(* PLC project Untitled3, Machine Expert Logic Builder V20.2.8.0, author Dylan *)
(* stored: creationDateTime 2023-03-14T07:56:13.4423497, version 0.0.0.0, modificationDateTime 2023-03-14T07:50:20.7728171 *)

{attribute 'qualified_only'}
{attribute 'strict'}
TYPE ET_9STATE_MONITORING : (STOPPED := 0, RUNNING := 1, STARTING := 2, STOPPING := 3, START_FAIL := 4, STOP_FAIL := 5, UNEXPECTED_START := 6, UNEXPECTED_STOP := 7, FIRE_STOP := 8, UNKNOWN := 9);
END_TYPE

{attribute 'qualified_only'}
{attribute 'strict'}
TYPE ET_ROOM_STATE : (DEPROX := 0, STANDBY := 1, ALARM := 2, ISOLATE := 3, POSITVE := 4);
END_TYPE

{attribute 'qualified_only'}
{attribute 'strict'}
TYPE ET_ROOM_MODE : (ISOLATION := 0, STANDBY := 1);
END_TYPE

PROGRAM RM59_STATUS
  VAR
    RM_MODE : ET_ROOM_MODE;
    ALARM_DELAY : TON;
    IS_ALARM : BOOL;
    TOF_BUZZER : TOF;
    RM_BUZZER_LOCAL : BOOL;
    IS_LOCAL_ALARM : BOOL;
    FB_ROOM_STATE_0 : FB_ROOM_STATE;
  END_VAR

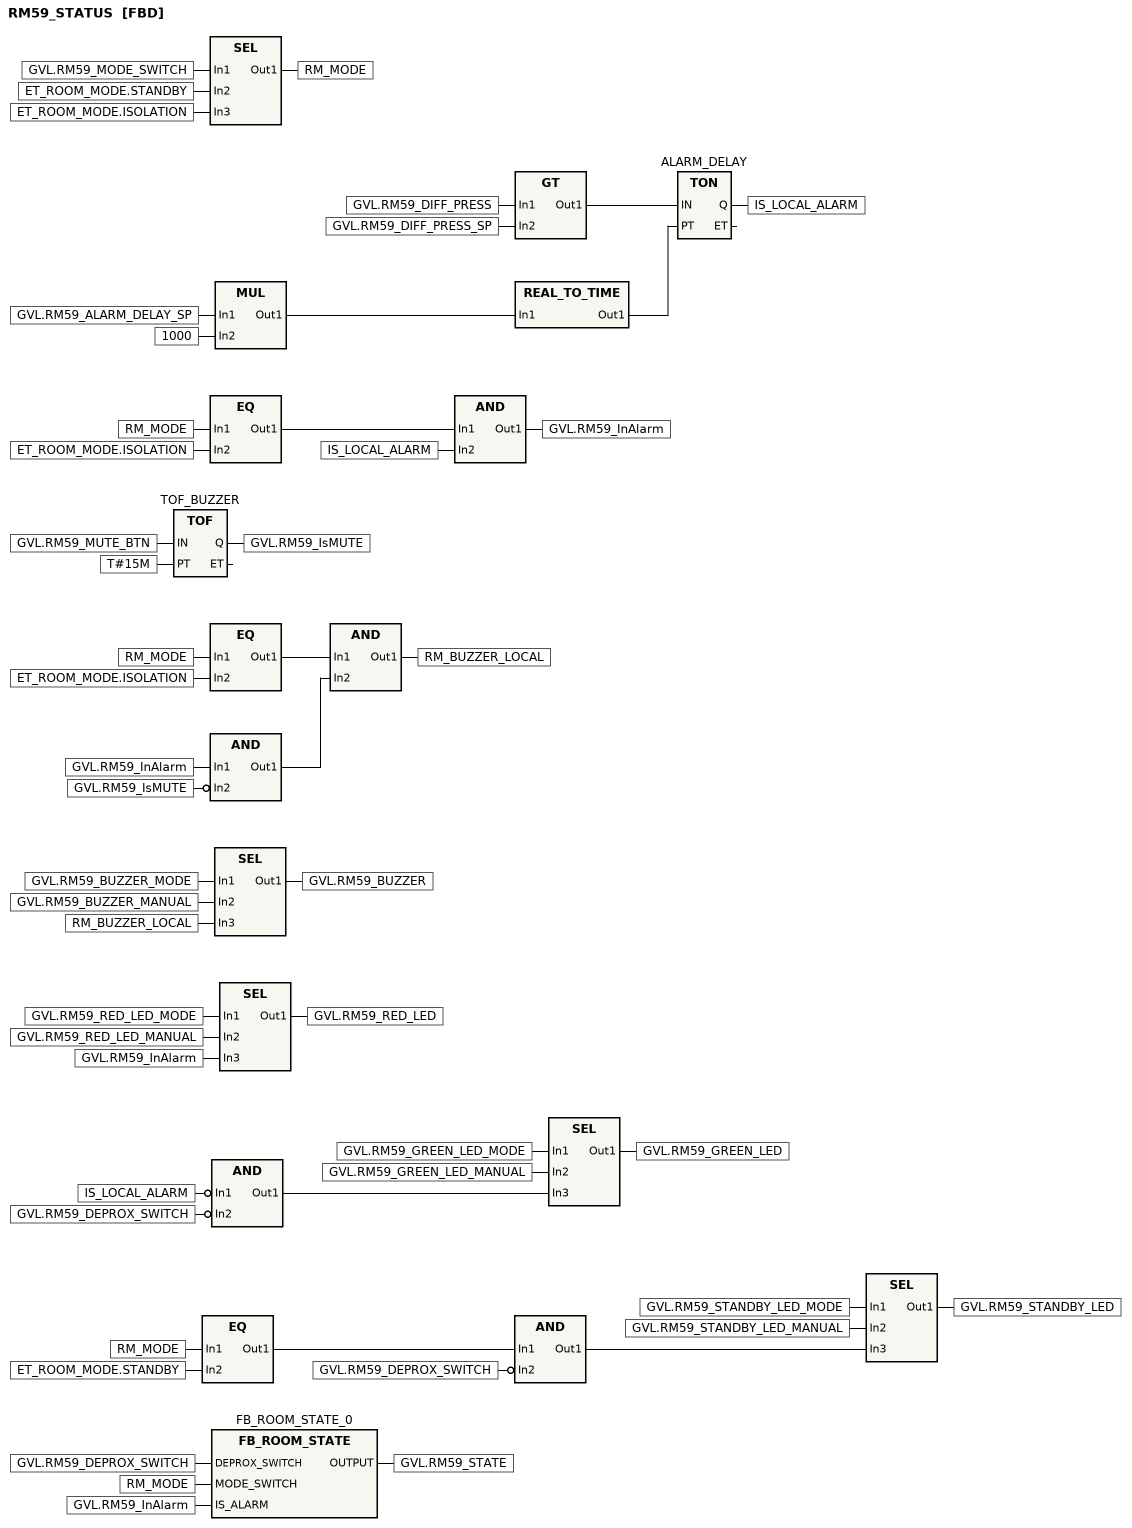
(* FBD diagram, written out as Structured Text *)
(* The mode switch located on the room alarm panel is to switch the room status between isolation mode and standby mode. *)
RM_MODE := SEL(GVL.RM59_MODE_SWITCH, ET_ROOM_MODE.STANDBY, ET_ROOM_MODE.ISOLATION);
(* generate alarms when RM DIFF PRESS >  RM DIFF PRESS SP.
the alarm will show on LED *)
ALARM_DELAY(IN := GVL.RM59_DIFF_PRESS > GVL.RM59_DIFF_PRESS_SP, PT := REAL_TO_TIME(GVL.RM59_ALARM_DELAY_SP * 1000));
IS_LOCAL_ALARM := ALARM_DELAY.Q;
(* ROOM IN ALARM *)
GVL.RM59_InAlarm := RM_MODE = ET_ROOM_MODE.ISOLATION AND IS_LOCAL_ALARM;
(* BUZZER
If the room is operating in isolation mode, the buzzer will activate until the panel RED button is pressed by an operator. If the room pressure remains outside of the acceptable range for a further 15 minutes, then the room buzzer will re-enable.

DISABLE BUZZER *)
TOF_BUZZER(IN := GVL.RM59_MUTE_BTN, PT := T#15M);
GVL.RM59_IsMUTE := TOF_BUZZER.Q;
(* BUZZER
If the room is operating in isolation mode, the buzzer will activate until the panel RED button is pressed by an operator. If the room pressure remains outside of the acceptable range for a further 15 minutes, then the room buzzer will re-enable. *)
RM_BUZZER_LOCAL := RM_MODE = ET_ROOM_MODE.ISOLATION AND GVL.RM59_InAlarm AND NOT GVL.RM59_IsMUTE;
(* AUTO/ MANUAL  MODE FROM BMS / BUZZER *)
GVL.RM59_BUZZER := SEL(GVL.RM59_BUZZER_MODE, GVL.RM59_BUZZER_MANUAL, RM_BUZZER_LOCAL);
(* AUTO/ MANUAL  MODE FROM BMS / RED LED *)
GVL.RM59_RED_LED := SEL(GVL.RM59_RED_LED_MODE, GVL.RM59_RED_LED_MANUAL, GVL.RM59_InAlarm);
(* AUTO/ MANUAL  MODE FROM BMS / GREEN LED *)
GVL.RM59_GREEN_LED := SEL(GVL.RM59_GREEN_LED_MODE, GVL.RM59_GREEN_LED_MANUAL, NOT IS_LOCAL_ALARM AND NOT GVL.RM59_DEPROX_SWITCH);
GVL.RM59_STANDBY_LED := SEL(GVL.RM59_STANDBY_LED_MODE, GVL.RM59_STANDBY_LED_MANUAL, RM_MODE = ET_ROOM_MODE.STANDBY AND NOT GVL.RM59_DEPROX_SWITCH);
(* ROOMT STATUS *)
FB_ROOM_STATE_0(DEPROX_SWITCH := GVL.RM59_DEPROX_SWITCH, MODE_SWITCH := RM_MODE, IS_ALARM := GVL.RM59_InAlarm);
GVL.RM59_STATE := FB_ROOM_STATE_0.OUTPUT;
END_PROGRAM

PROGRAM RM51_DEPROX
  VAR
    ENABLE_BLINKING : BOOL;
    FB_PULSE_GENERATOR_0 : FB_PULSE_GENERATOR;
  END_VAR

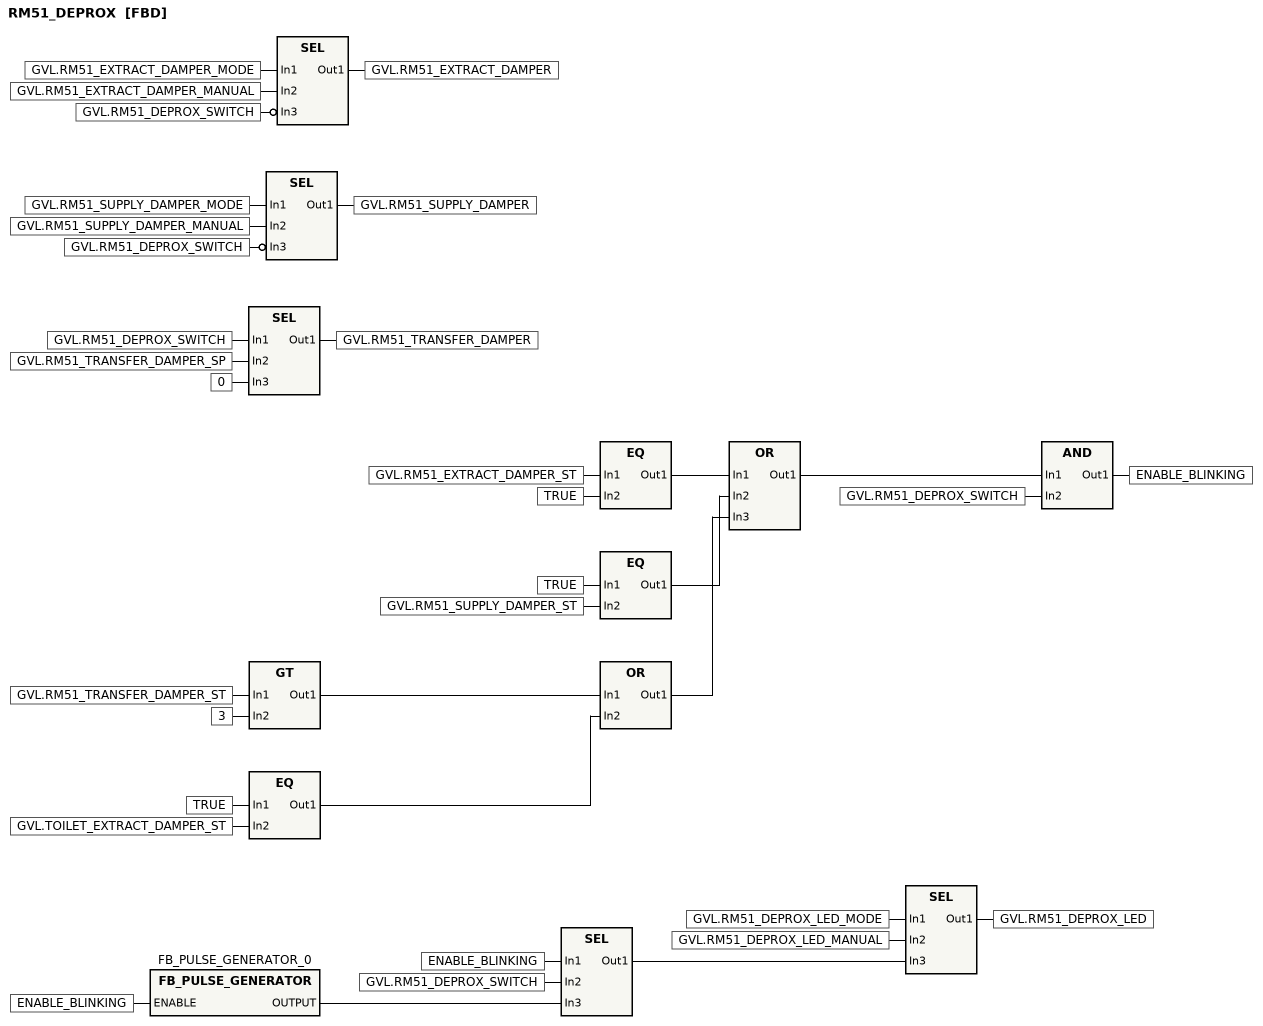
(* FBD diagram, written out as Structured Text *)
(* Return Air Damper - close damper in deprox mode

Deprox Switch. 0=normal 1=deprox *)
GVL.RM51_EXTRACT_DAMPER := SEL(GVL.RM51_EXTRACT_DAMPER_MODE, GVL.RM51_EXTRACT_DAMPER_MANUAL, NOT GVL.RM51_DEPROX_SWITCH);
(* Supply Air Damper - close damper in deprox mode

Deprox Switch. 0=normal 1=deprox *)
GVL.RM51_SUPPLY_DAMPER := SEL(GVL.RM51_SUPPLY_DAMPER_MODE, GVL.RM51_SUPPLY_DAMPER_MANUAL, NOT GVL.RM51_DEPROX_SWITCH);
(* Transfer Damper - close damper in deprox mode

Deprox Switch. 0=normal 1=deprox *)
GVL.RM51_TRANSFER_DAMPER := SEL(GVL.RM51_DEPROX_SWITCH, GVL.RM51_TRANSFER_DAMPER_SP, 0);
(* enable blinking when the room dampers are driving closed *)
ENABLE_BLINKING := (GVL.RM51_EXTRACT_DAMPER_ST = TRUE OR TRUE = GVL.RM51_SUPPLY_DAMPER_ST OR GVL.RM51_TRANSFER_DAMPER_ST > 3 OR TRUE = GVL.TOILET_EXTRACT_DAMPER_ST) AND GVL.RM51_DEPROX_SWITCH;
(* DEPROX LED *)
FB_PULSE_GENERATOR_0(ENABLE := ENABLE_BLINKING);
GVL.RM51_DEPROX_LED := SEL(GVL.RM51_DEPROX_LED_MODE, GVL.RM51_DEPROX_LED_MANUAL, SEL(ENABLE_BLINKING, GVL.RM51_DEPROX_SWITCH, FB_PULSE_GENERATOR_0.OUTPUT));
END_PROGRAM

FUNCTION_BLOCK FB_2STAGES_DUTY
  VAR_INPUT
    isFAN1_FAULT : BOOL;
    isFAN2_FAULT : BOOL;
    STANDBY_FAN : INT := 1;
    FAN_SPD : REAL;
  END_VAR
  VAR_OUTPUT
    FAN1_ENABLE : BOOL;
    FAN2_ENABLE : BOOL;
    FAN1_SPD : REAL;
    FAN2_SPD : REAL;
  END_VAR

                    IF (STANDBY_FAN = 1) THEN
	IF(isFAN2_FAULT) THEN
		FAN1_ENABLE := TRUE;
		FAN1_SPD := FAN_SPD;
	ELSE
		FAN1_ENABLE := FALSE;
		FAN1_SPD := 0.0;
	END_IF;
	FAN2_ENABLE := TRUE;
	FAN2_SPD := FAN_SPD;
ELSIF (STANDBY_FAN = 2) THEN
	IF(isFAN1_FAULT) THEN
		FAN2_ENABLE := TRUE;
		FAN2_SPD := FAN_SPD;
	ELSE
		FAN2_ENABLE := FALSE;
		FAN2_SPD := 0.0;
	END_IF;
	FAN1_ENABLE := TRUE;
	FAN1_SPD := FAN_SPD;
END_IF;

                  
END_FUNCTION_BLOCK

PROGRAM RM119_DEPROX
  VAR
    ENABLE_BLINKING : BOOL;
    FB_PULSE_GENERATOR_0 : FB_PULSE_GENERATOR;
  END_VAR

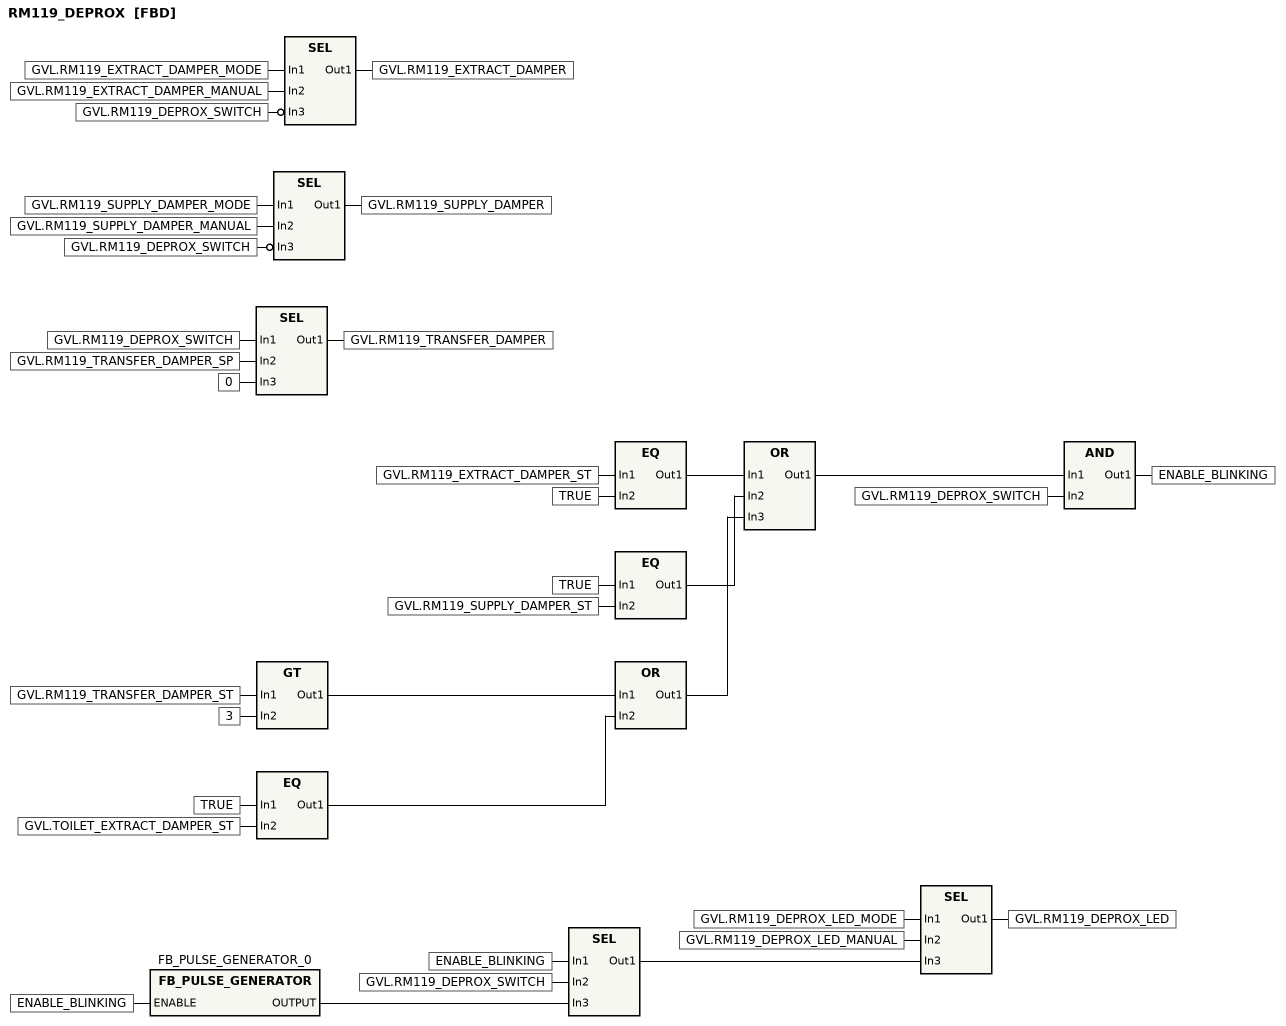
(* FBD diagram, written out as Structured Text *)
(* Return Air Damper - close damper in deprox mode

Deprox Switch. 0=normal 1=deprox *)
GVL.RM119_EXTRACT_DAMPER := SEL(GVL.RM119_EXTRACT_DAMPER_MODE, GVL.RM119_EXTRACT_DAMPER_MANUAL, NOT GVL.RM119_DEPROX_SWITCH);
(* Supply Air Damper - close damper in deprox mode

Deprox Switch. 0=normal 1=deprox *)
GVL.RM119_SUPPLY_DAMPER := SEL(GVL.RM119_SUPPLY_DAMPER_MODE, GVL.RM119_SUPPLY_DAMPER_MANUAL, NOT GVL.RM119_DEPROX_SWITCH);
(* Transfer Damper - close damper in deprox mode

Deprox Switch. 0=normal 1=deprox *)
GVL.RM119_TRANSFER_DAMPER := SEL(GVL.RM119_DEPROX_SWITCH, GVL.RM119_TRANSFER_DAMPER_SP, 0);
(* enable blinking when the room dampers are driving closed *)
ENABLE_BLINKING := (GVL.RM119_EXTRACT_DAMPER_ST = TRUE OR TRUE = GVL.RM119_SUPPLY_DAMPER_ST OR GVL.RM119_TRANSFER_DAMPER_ST > 3 OR TRUE = GVL.TOILET_EXTRACT_DAMPER_ST) AND GVL.RM119_DEPROX_SWITCH;
(* DEPROX LED *)
FB_PULSE_GENERATOR_0(ENABLE := ENABLE_BLINKING);
GVL.RM119_DEPROX_LED := SEL(GVL.RM119_DEPROX_LED_MODE, GVL.RM119_DEPROX_LED_MANUAL, SEL(ENABLE_BLINKING, GVL.RM119_DEPROX_SWITCH, FB_PULSE_GENERATOR_0.OUTPUT));
END_PROGRAM

FUNCTION_BLOCK FB_DUTYTRIGGER
  VAR_INPUT
    INPUT : BOOL;
    MAX_STAGE : INT := 2;
    CURRENT_STAGE : INT;
  END_VAR
  VAR_OUTPUT
    RESULT : INT;
  END_VAR

                    IF(INPUT) THEN
	RESULT := CURRENT_STAGE + 1;
END_IF;

IF(RESULT > MAX_STAGE) OR (RESULT <= 0) THEN
	RESULT:= 1;
END_IF;


                  
END_FUNCTION_BLOCK

PROGRAM RM52_DEPROX
  VAR
    ENABLE_BLINKING : BOOL;
    FB_PULSE_GENERATOR_0 : FB_PULSE_GENERATOR;
  END_VAR

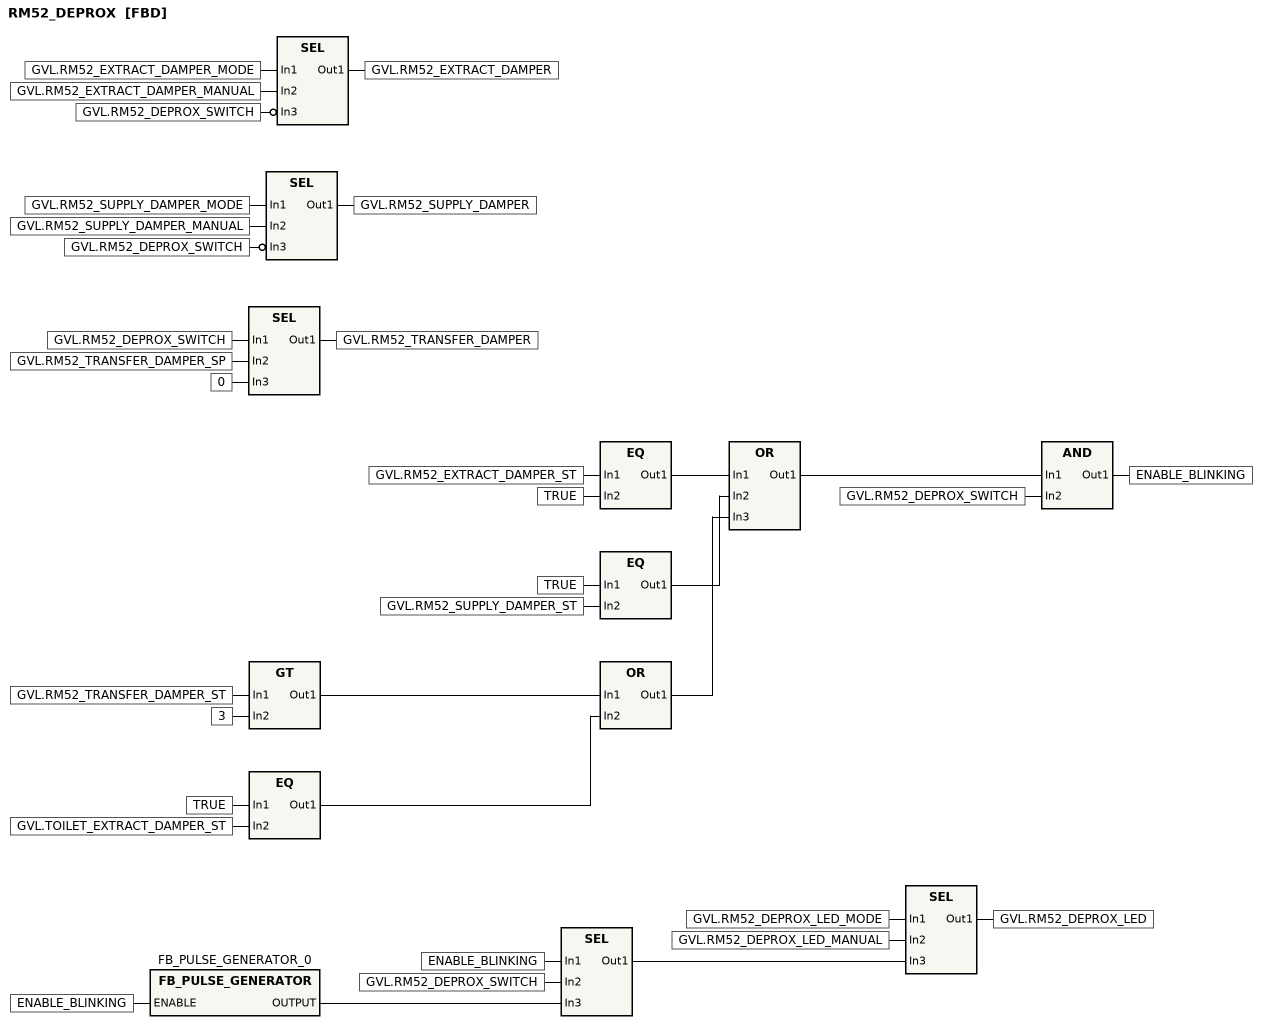
(* FBD diagram, written out as Structured Text *)
(* Return Air Damper - close damper in deprox mode

Deprox Switch. 0=normal 1=deprox *)
GVL.RM52_EXTRACT_DAMPER := SEL(GVL.RM52_EXTRACT_DAMPER_MODE, GVL.RM52_EXTRACT_DAMPER_MANUAL, NOT GVL.RM52_DEPROX_SWITCH);
(* Supply Air Damper - close damper in deprox mode

Deprox Switch. 0=normal 1=deprox *)
GVL.RM52_SUPPLY_DAMPER := SEL(GVL.RM52_SUPPLY_DAMPER_MODE, GVL.RM52_SUPPLY_DAMPER_MANUAL, NOT GVL.RM52_DEPROX_SWITCH);
(* Transfer Damper - close damper in deprox mode

Deprox Switch. 0=normal 1=deprox *)
GVL.RM52_TRANSFER_DAMPER := SEL(GVL.RM52_DEPROX_SWITCH, GVL.RM52_TRANSFER_DAMPER_SP, 0);
(* enable blinking when the room dampers are driving closed *)
ENABLE_BLINKING := (GVL.RM52_EXTRACT_DAMPER_ST = TRUE OR TRUE = GVL.RM52_SUPPLY_DAMPER_ST OR GVL.RM52_TRANSFER_DAMPER_ST > 3 OR TRUE = GVL.TOILET_EXTRACT_DAMPER_ST) AND GVL.RM52_DEPROX_SWITCH;
(* DEPROX LED *)
FB_PULSE_GENERATOR_0(ENABLE := ENABLE_BLINKING);
GVL.RM52_DEPROX_LED := SEL(GVL.RM52_DEPROX_LED_MODE, GVL.RM52_DEPROX_LED_MANUAL, SEL(ENABLE_BLINKING, GVL.RM52_DEPROX_SWITCH, FB_PULSE_GENERATOR_0.OUTPUT));
END_PROGRAM

PROGRAM RM53_DEPROX
  VAR
    ENABLE_BLINKING : BOOL;
    FB_PULSE_GENERATOR_0 : FB_PULSE_GENERATOR;
  END_VAR

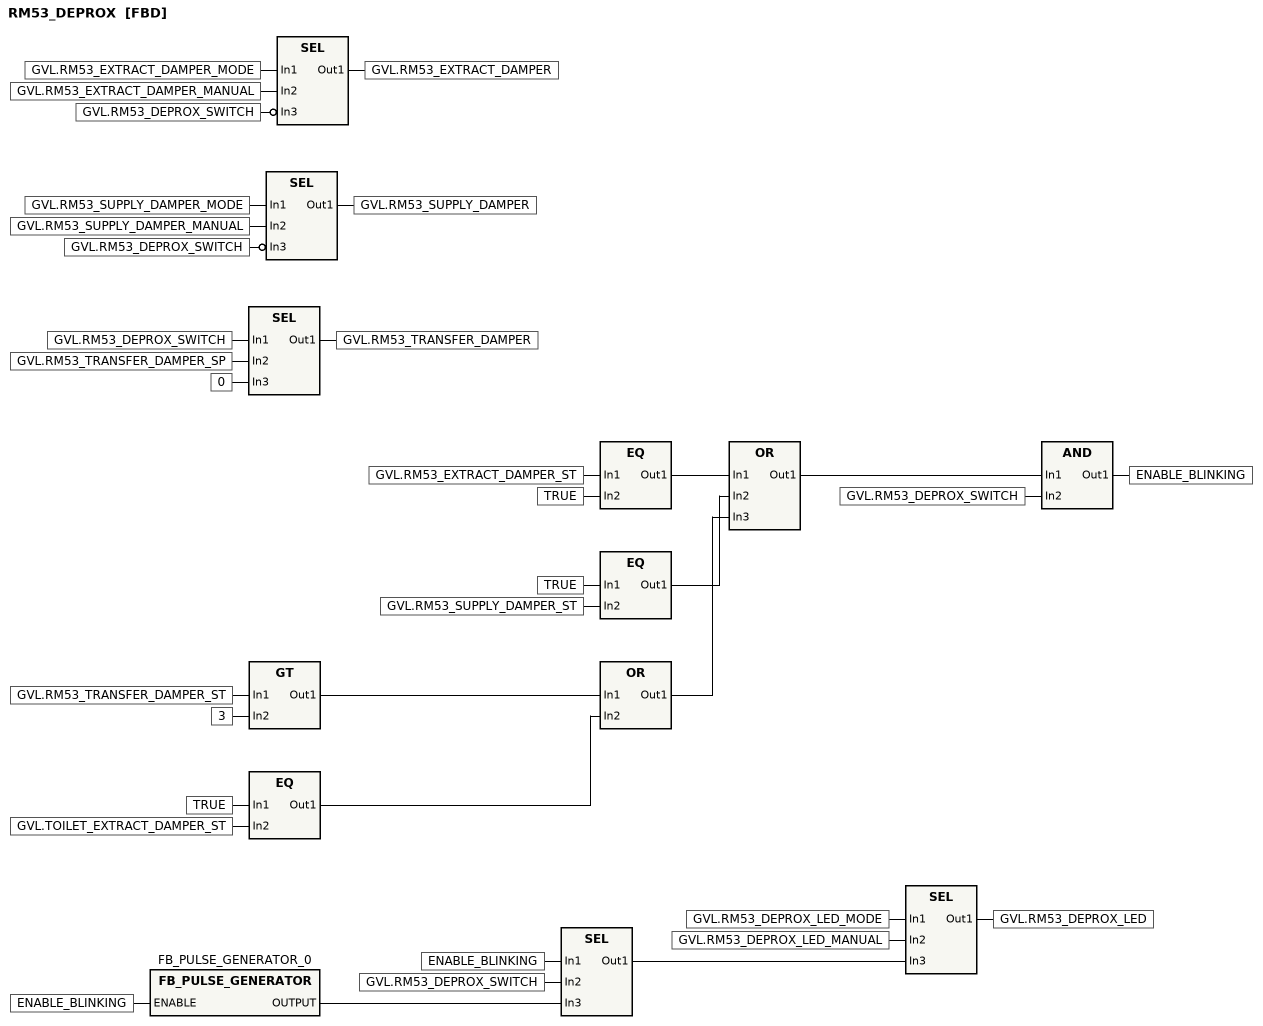
(* FBD diagram, written out as Structured Text *)
(* Return Air Damper - close damper in deprox mode

Deprox Switch. 0=normal 1=deprox *)
GVL.RM53_EXTRACT_DAMPER := SEL(GVL.RM53_EXTRACT_DAMPER_MODE, GVL.RM53_EXTRACT_DAMPER_MANUAL, NOT GVL.RM53_DEPROX_SWITCH);
(* Supply Air Damper - close damper in deprox mode

Deprox Switch. 0=normal 1=deprox *)
GVL.RM53_SUPPLY_DAMPER := SEL(GVL.RM53_SUPPLY_DAMPER_MODE, GVL.RM53_SUPPLY_DAMPER_MANUAL, NOT GVL.RM53_DEPROX_SWITCH);
(* Transfer Damper - close damper in deprox mode

Deprox Switch. 0=normal 1=deprox *)
GVL.RM53_TRANSFER_DAMPER := SEL(GVL.RM53_DEPROX_SWITCH, GVL.RM53_TRANSFER_DAMPER_SP, 0);
(* enable blinking when the room dampers are driving closed *)
ENABLE_BLINKING := (GVL.RM53_EXTRACT_DAMPER_ST = TRUE OR TRUE = GVL.RM53_SUPPLY_DAMPER_ST OR GVL.RM53_TRANSFER_DAMPER_ST > 3 OR TRUE = GVL.TOILET_EXTRACT_DAMPER_ST) AND GVL.RM53_DEPROX_SWITCH;
(* DEPROX LED *)
FB_PULSE_GENERATOR_0(ENABLE := ENABLE_BLINKING);
GVL.RM53_DEPROX_LED := SEL(GVL.RM53_DEPROX_LED_MODE, GVL.RM53_DEPROX_LED_MANUAL, SEL(ENABLE_BLINKING, GVL.RM53_DEPROX_SWITCH, FB_PULSE_GENERATOR_0.OUTPUT));
END_PROGRAM

FUNCTION_BLOCK FB_3STAGES_DUTY
  VAR_INPUT
    isFAN1_FAULT : BOOL;
    isFAN2_FAULT : BOOL;
    isFAN3_FAULT : BOOL;
    STANDBY_FAN : INT := 1;
    FAN_SPD : REAL;
  END_VAR
  VAR_OUTPUT
    FAN1_ENABLE : BOOL;
    FAN2_ENABLE : BOOL;
    FAN3_ENABLE : BOOL;
    FAN1_SPD : REAL;
    FAN2_SPD : REAL;
    FAN3_SPD : REAL;
  END_VAR

                    IF (STANDBY_FAN = 1) THEN
	IF(isFAN2_FAULT OR isFAN3_FAULT) THEN
		FAN1_ENABLE := TRUE;
		FAN1_SPD := FAN_SPD;
	ELSE
		FAN1_ENABLE := FALSE;
		FAN1_SPD := 0.0;
	END_IF;
	FAN2_ENABLE := TRUE;
	FAN3_ENABLE := TRUE;
	FAN2_SPD := FAN_SPD;
	FAN3_SPD := FAN_SPD;
ELSIF (STANDBY_FAN = 2) THEN
	IF(isFAN1_FAULT OR isFAN3_FAULT) THEN
		FAN2_ENABLE := TRUE;
		FAN2_SPD := FAN_SPD;
	ELSE
		FAN2_ENABLE := FALSE;
		FAN2_SPD := 0.0;
	END_IF;
	FAN1_ENABLE := TRUE;
	FAN3_ENABLE := TRUE;
	FAN1_SPD := FAN_SPD;
	FAN3_SPD := FAN_SPD;
ELSIF (STANDBY_FAN = 3) THEN
	IF(isFAN1_FAULT OR isFAN2_FAULT) THEN
		FAN3_ENABLE := TRUE;
		FAN3_SPD := FAN_SPD;
	ELSE
		FAN3_ENABLE := FALSE;
		FAN3_SPD := 0.0;
	END_IF;
	FAN1_ENABLE := TRUE;
	FAN2_ENABLE := TRUE;
	FAN1_SPD := FAN_SPD;
	FAN2_SPD := FAN_SPD;
END_IF;

                  
END_FUNCTION_BLOCK

PROGRAM RM119_STATUS
  VAR
    RM_MODE : ET_ROOM_MODE;
    ALARM_DELAY : TON;
    IS_ALARM : BOOL;
    TOF_BUZZER : TOF;
    RM_BUZZER_LOCAL : BOOL;
    IS_LOCAL_ALARM : BOOL;
    FB_ROOM_STATE_0 : FB_ROOM_STATE;
  END_VAR

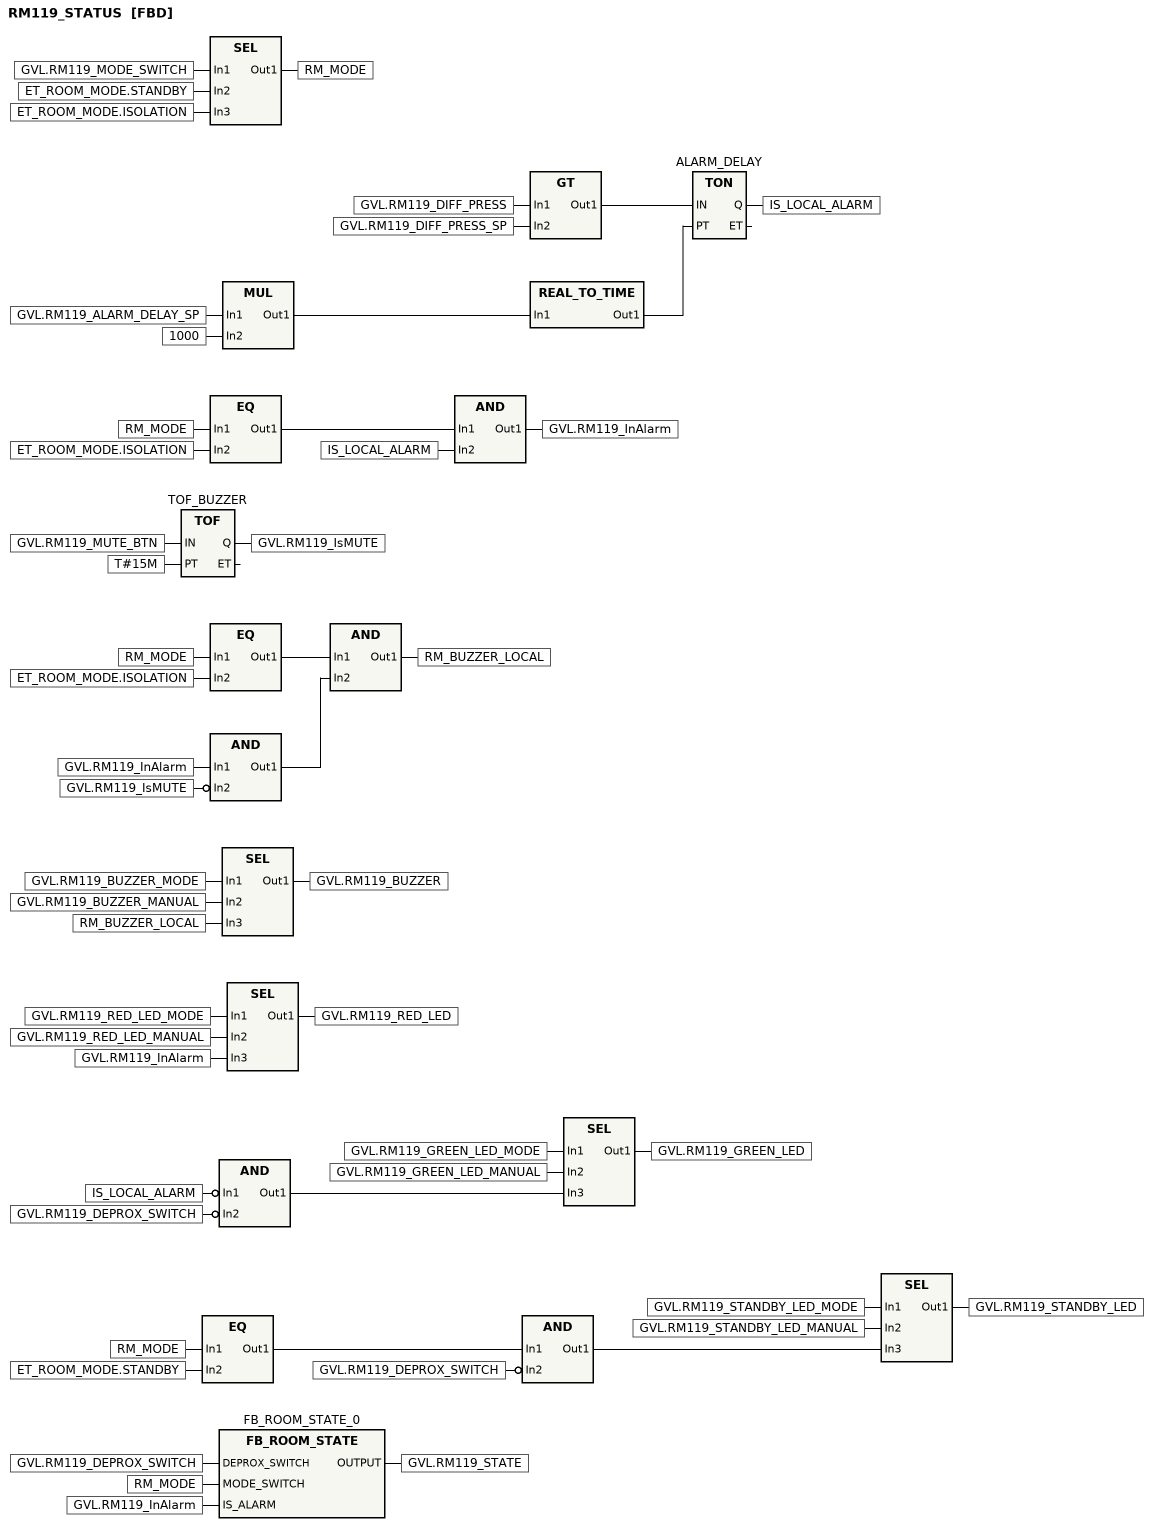
(* FBD diagram, written out as Structured Text *)
(* The mode switch located on the room alarm panel is to switch the room status between isolation mode and standby mode. *)
RM_MODE := SEL(GVL.RM119_MODE_SWITCH, ET_ROOM_MODE.STANDBY, ET_ROOM_MODE.ISOLATION);
(* generate alarms when RM DIFF PRESS >  RM DIFF PRESS SP.
the alarm will show on LED *)
ALARM_DELAY(IN := GVL.RM119_DIFF_PRESS > GVL.RM119_DIFF_PRESS_SP, PT := REAL_TO_TIME(GVL.RM119_ALARM_DELAY_SP * 1000));
IS_LOCAL_ALARM := ALARM_DELAY.Q;
(* ROOM IN ALARM *)
GVL.RM119_InAlarm := RM_MODE = ET_ROOM_MODE.ISOLATION AND IS_LOCAL_ALARM;
(* BUZZER
If the room is operating in isolation mode, the buzzer will activate until the panel RED button is pressed by an operator. If the room pressure remains outside of the acceptable range for a further 15 minutes, then the room buzzer will re-enable.

DISABLE BUZZER *)
TOF_BUZZER(IN := GVL.RM119_MUTE_BTN, PT := T#15M);
GVL.RM119_IsMUTE := TOF_BUZZER.Q;
(* BUZZER
If the room is operating in isolation mode, the buzzer will activate until the panel RED button is pressed by an operator. If the room pressure remains outside of the acceptable range for a further 15 minutes, then the room buzzer will re-enable. *)
RM_BUZZER_LOCAL := RM_MODE = ET_ROOM_MODE.ISOLATION AND GVL.RM119_InAlarm AND NOT GVL.RM119_IsMUTE;
(* AUTO/ MANUAL  MODE FROM BMS / BUZZER *)
GVL.RM119_BUZZER := SEL(GVL.RM119_BUZZER_MODE, GVL.RM119_BUZZER_MANUAL, RM_BUZZER_LOCAL);
(* AUTO/ MANUAL  MODE FROM BMS / RED LED *)
GVL.RM119_RED_LED := SEL(GVL.RM119_RED_LED_MODE, GVL.RM119_RED_LED_MANUAL, GVL.RM119_InAlarm);
(* AUTO/ MANUAL  MODE FROM BMS / GREEN LED *)
GVL.RM119_GREEN_LED := SEL(GVL.RM119_GREEN_LED_MODE, GVL.RM119_GREEN_LED_MANUAL, NOT IS_LOCAL_ALARM AND NOT GVL.RM119_DEPROX_SWITCH);
GVL.RM119_STANDBY_LED := SEL(GVL.RM119_STANDBY_LED_MODE, GVL.RM119_STANDBY_LED_MANUAL, RM_MODE = ET_ROOM_MODE.STANDBY AND NOT GVL.RM119_DEPROX_SWITCH);
(* ROOMT STATUS *)
FB_ROOM_STATE_0(DEPROX_SWITCH := GVL.RM119_DEPROX_SWITCH, MODE_SWITCH := RM_MODE, IS_ALARM := GVL.RM119_InAlarm);
GVL.RM119_STATE := FB_ROOM_STATE_0.OUTPUT;
END_PROGRAM

PROGRAM RM71_DEPROX
  VAR
    ENABLE_BLINKING : BOOL;
    FB_PULSE_GENERATOR_0 : FB_PULSE_GENERATOR;
  END_VAR

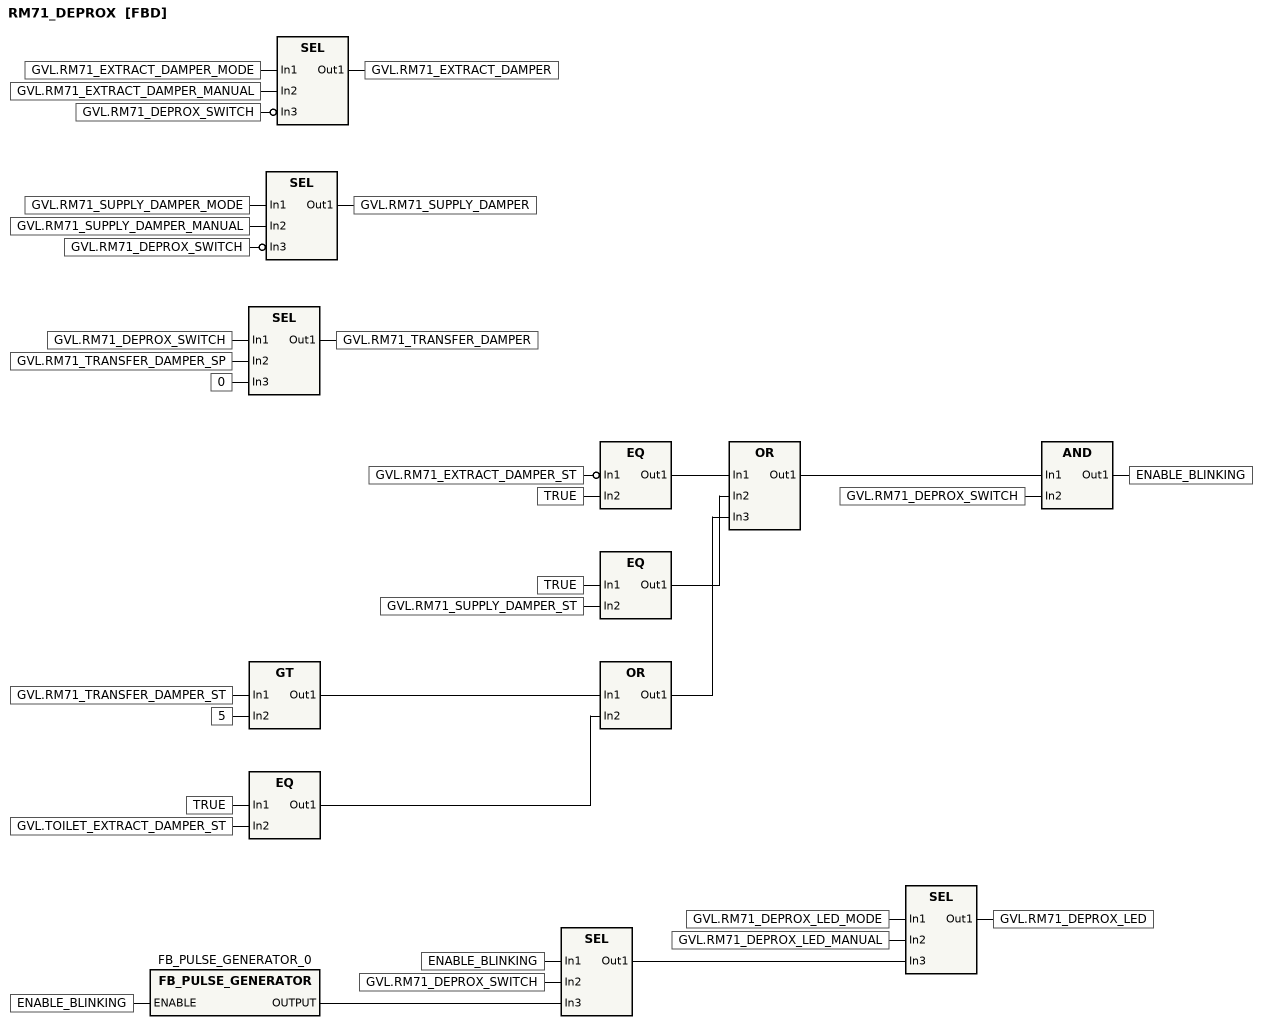
(* FBD diagram, written out as Structured Text *)
(* Return Air Damper - close damper in deprox mode

Deprox Switch. 0=normal 1=deprox *)
GVL.RM71_EXTRACT_DAMPER := SEL(GVL.RM71_EXTRACT_DAMPER_MODE, GVL.RM71_EXTRACT_DAMPER_MANUAL, NOT GVL.RM71_DEPROX_SWITCH);
(* Supply Air Damper - close damper in deprox mode

Deprox Switch. 0=normal 1=deprox *)
GVL.RM71_SUPPLY_DAMPER := SEL(GVL.RM71_SUPPLY_DAMPER_MODE, GVL.RM71_SUPPLY_DAMPER_MANUAL, NOT GVL.RM71_DEPROX_SWITCH);
(* Transfer Damper - close damper in deprox mode

Deprox Switch. 0=normal 1=deprox *)
GVL.RM71_TRANSFER_DAMPER := SEL(GVL.RM71_DEPROX_SWITCH, GVL.RM71_TRANSFER_DAMPER_SP, 0);
(* enable blinking when the room dampers are driving closed *)
ENABLE_BLINKING := (NOT GVL.RM71_EXTRACT_DAMPER_ST = TRUE OR TRUE = GVL.RM71_SUPPLY_DAMPER_ST OR GVL.RM71_TRANSFER_DAMPER_ST > 5 OR TRUE = GVL.TOILET_EXTRACT_DAMPER_ST) AND GVL.RM71_DEPROX_SWITCH;
(* DEPROX LED *)
FB_PULSE_GENERATOR_0(ENABLE := ENABLE_BLINKING);
GVL.RM71_DEPROX_LED := SEL(GVL.RM71_DEPROX_LED_MODE, GVL.RM71_DEPROX_LED_MANUAL, SEL(ENABLE_BLINKING, GVL.RM71_DEPROX_SWITCH, FB_PULSE_GENERATOR_0.OUTPUT));
END_PROGRAM

FUNCTION_BLOCK FB_0_10V_TO_2_10V_OUTPUT
  VAR_OUTPUT
    OUT_PRCT : REAL;  (* 0-10V = 0-100% *)
  END_VAR
  VAR_INPUT
    IN_PRCT : REAL;  (* 2-10V = 0-100% *)
  END_VAR

                    OUT_PRCT := ((IN_PRCT * 0.08) + 2) * 10;
                  
END_FUNCTION_BLOCK

PROGRAM RM52_STATUS
  VAR
    RM_MODE : ET_ROOM_MODE;
    ALARM_DELAY : TON;
    IS_ALARM : BOOL;
    TOF_BUZZER : TOF;
    RM_BUZZER_LOCAL : BOOL;
    IS_LOCAL_ALARM : BOOL;
    FB_ROOM_STATE_0 : FB_ROOM_STATE;
  END_VAR

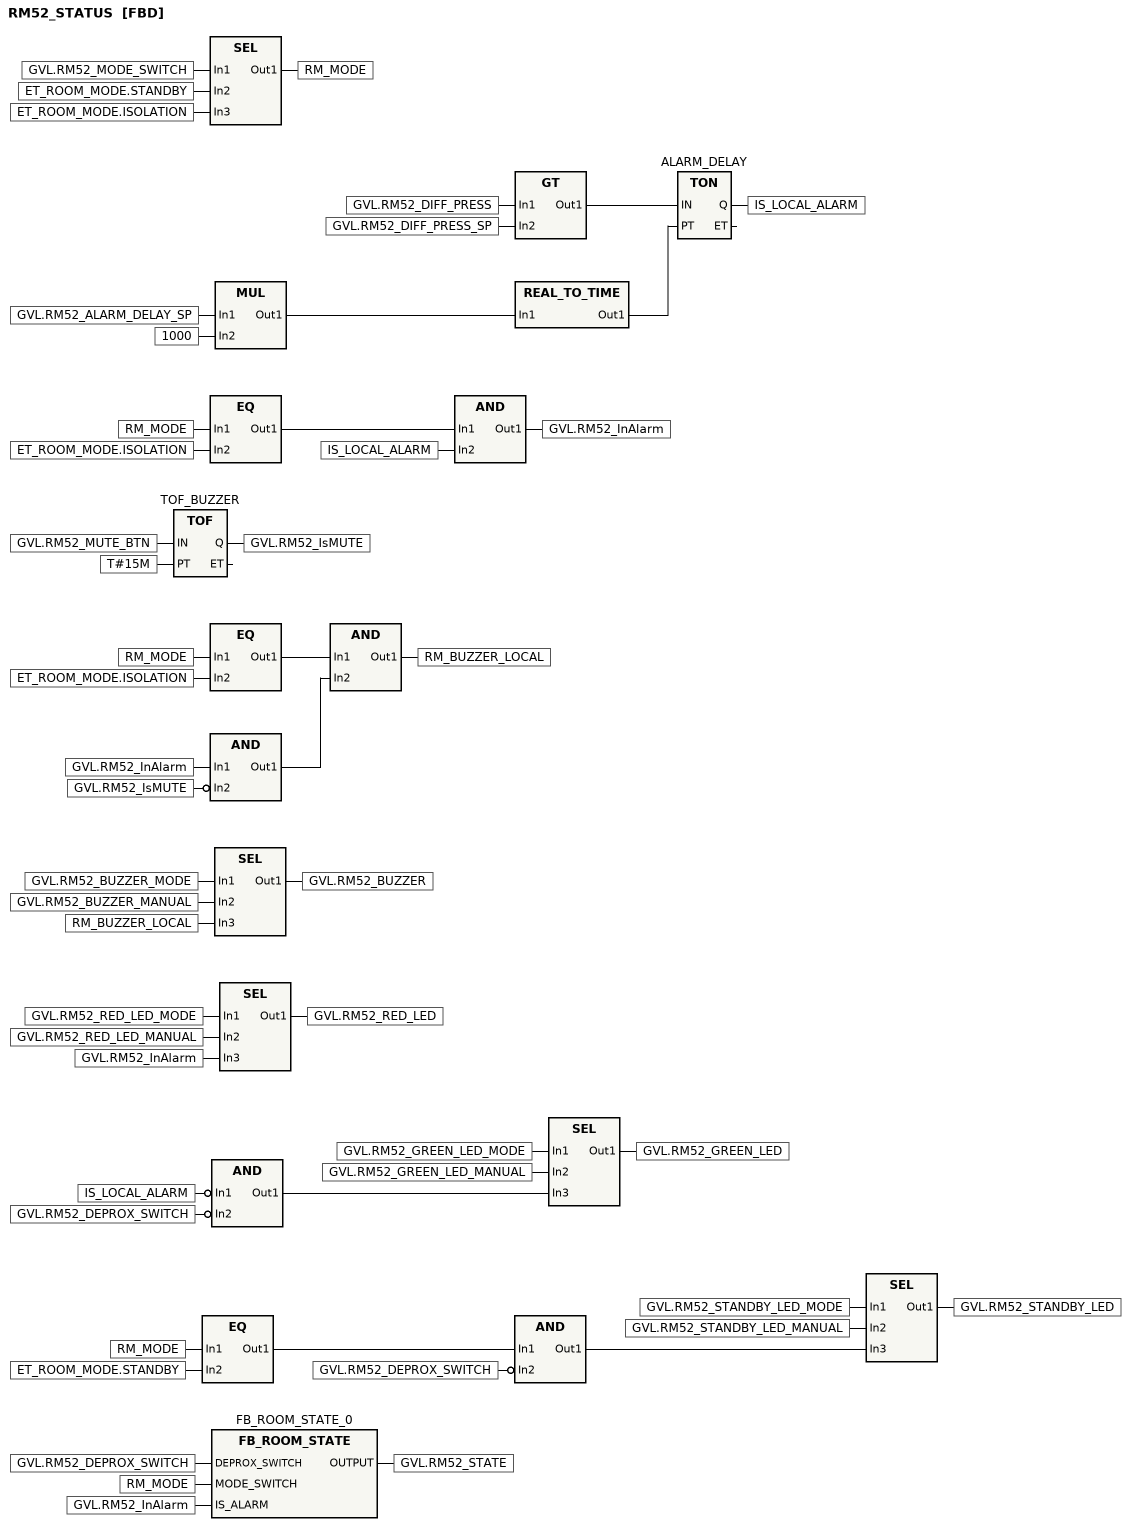
(* FBD diagram, written out as Structured Text *)
(* The mode switch located on the room alarm panel is to switch the room status between isolation mode and standby mode. *)
RM_MODE := SEL(GVL.RM52_MODE_SWITCH, ET_ROOM_MODE.STANDBY, ET_ROOM_MODE.ISOLATION);
(* generate alarms when RM DIFF PRESS >  RM DIFF PRESS SP.
the alarm will show on LED *)
ALARM_DELAY(IN := GVL.RM52_DIFF_PRESS > GVL.RM52_DIFF_PRESS_SP, PT := REAL_TO_TIME(GVL.RM52_ALARM_DELAY_SP * 1000));
IS_LOCAL_ALARM := ALARM_DELAY.Q;
(* ROOM IN ALARM *)
GVL.RM52_InAlarm := RM_MODE = ET_ROOM_MODE.ISOLATION AND IS_LOCAL_ALARM;
(* BUZZER
If the room is operating in isolation mode, the buzzer will activate until the panel RED button is pressed by an operator. If the room pressure remains outside of the acceptable range for a further 15 minutes, then the room buzzer will re-enable.

DISABLE BUZZER *)
TOF_BUZZER(IN := GVL.RM52_MUTE_BTN, PT := T#15M);
GVL.RM52_IsMUTE := TOF_BUZZER.Q;
(* BUZZER
If the room is operating in isolation mode, the buzzer will activate until the panel RED button is pressed by an operator. If the room pressure remains outside of the acceptable range for a further 15 minutes, then the room buzzer will re-enable. *)
RM_BUZZER_LOCAL := RM_MODE = ET_ROOM_MODE.ISOLATION AND GVL.RM52_InAlarm AND NOT GVL.RM52_IsMUTE;
(* AUTO/ MANUAL  MODE FROM BMS / BUZZER *)
GVL.RM52_BUZZER := SEL(GVL.RM52_BUZZER_MODE, GVL.RM52_BUZZER_MANUAL, RM_BUZZER_LOCAL);
(* AUTO/ MANUAL  MODE FROM BMS / RED LED *)
GVL.RM52_RED_LED := SEL(GVL.RM52_RED_LED_MODE, GVL.RM52_RED_LED_MANUAL, GVL.RM52_InAlarm);
(* AUTO/ MANUAL  MODE FROM BMS / GREEN LED *)
GVL.RM52_GREEN_LED := SEL(GVL.RM52_GREEN_LED_MODE, GVL.RM52_GREEN_LED_MANUAL, NOT IS_LOCAL_ALARM AND NOT GVL.RM52_DEPROX_SWITCH);
GVL.RM52_STANDBY_LED := SEL(GVL.RM52_STANDBY_LED_MODE, GVL.RM52_STANDBY_LED_MANUAL, RM_MODE = ET_ROOM_MODE.STANDBY AND NOT GVL.RM52_DEPROX_SWITCH);
(* ROOMT STATUS *)
FB_ROOM_STATE_0(DEPROX_SWITCH := GVL.RM52_DEPROX_SWITCH, MODE_SWITCH := RM_MODE, IS_ALARM := GVL.RM52_InAlarm);
GVL.RM52_STATE := FB_ROOM_STATE_0.OUTPUT;
END_PROGRAM

PROGRAM RM44_3_STATUS
  VAR
    RM_MODE : ET_ROOM_MODE;
    ALARM_DELAY : TON;
    IS_ALARM : BOOL;
    TOF_BUZZER : TOF;
    RM_BUZZER_LOCAL : BOOL;
    IS_LOCAL_ALARM : BOOL;
    FB_ROOM_STATE_0 : FB_ROOM_STATE;
  END_VAR

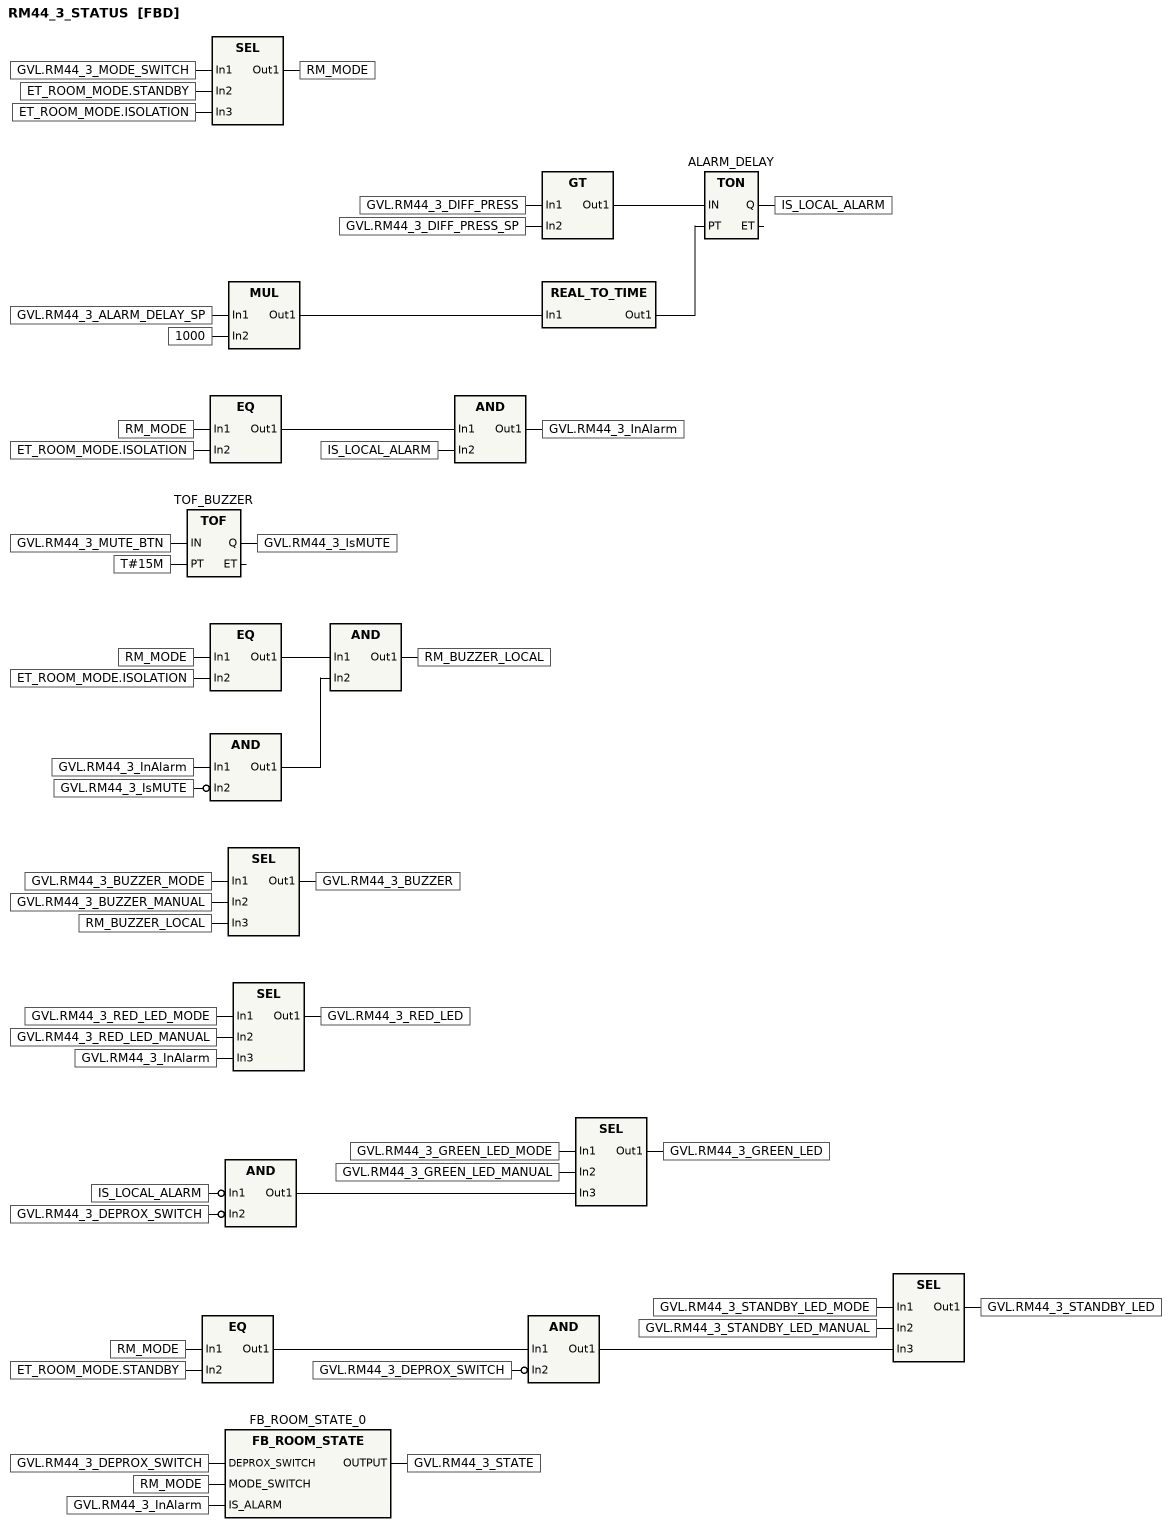
(* FBD diagram, written out as Structured Text *)
(* The mode switch located on the room alarm panel is to switch the room status between isolation mode and standby mode. *)
RM_MODE := SEL(GVL.RM44_3_MODE_SWITCH, ET_ROOM_MODE.STANDBY, ET_ROOM_MODE.ISOLATION);
(* generate alarms when RM DIFF PRESS >  RM DIFF PRESS SP.
the alarm will show on LED *)
ALARM_DELAY(IN := GVL.RM44_3_DIFF_PRESS > GVL.RM44_3_DIFF_PRESS_SP, PT := REAL_TO_TIME(GVL.RM44_3_ALARM_DELAY_SP * 1000));
IS_LOCAL_ALARM := ALARM_DELAY.Q;
(* ROOM IN ALARM *)
GVL.RM44_3_InAlarm := RM_MODE = ET_ROOM_MODE.ISOLATION AND IS_LOCAL_ALARM;
(* BUZZER
If the room is operating in isolation mode, the buzzer will activate until the panel RED button is pressed by an operator. If the room pressure remains outside of the acceptable range for a further 15 minutes, then the room buzzer will re-enable.

DISABLE BUZZER *)
TOF_BUZZER(IN := GVL.RM44_3_MUTE_BTN, PT := T#15M);
GVL.RM44_3_IsMUTE := TOF_BUZZER.Q;
(* BUZZER
If the room is operating in isolation mode, the buzzer will activate until the panel RED button is pressed by an operator. If the room pressure remains outside of the acceptable range for a further 15 minutes, then the room buzzer will re-enable. *)
RM_BUZZER_LOCAL := RM_MODE = ET_ROOM_MODE.ISOLATION AND GVL.RM44_3_InAlarm AND NOT GVL.RM44_3_IsMUTE;
(* AUTO/ MANUAL  MODE FROM BMS / BUZZER *)
GVL.RM44_3_BUZZER := SEL(GVL.RM44_3_BUZZER_MODE, GVL.RM44_3_BUZZER_MANUAL, RM_BUZZER_LOCAL);
(* AUTO/ MANUAL  MODE FROM BMS / RED LED *)
GVL.RM44_3_RED_LED := SEL(GVL.RM44_3_RED_LED_MODE, GVL.RM44_3_RED_LED_MANUAL, GVL.RM44_3_InAlarm);
(* AUTO/ MANUAL  MODE FROM BMS / GREEN LED *)
GVL.RM44_3_GREEN_LED := SEL(GVL.RM44_3_GREEN_LED_MODE, GVL.RM44_3_GREEN_LED_MANUAL, NOT IS_LOCAL_ALARM AND NOT GVL.RM44_3_DEPROX_SWITCH);
GVL.RM44_3_STANDBY_LED := SEL(GVL.RM44_3_STANDBY_LED_MODE, GVL.RM44_3_STANDBY_LED_MANUAL, RM_MODE = ET_ROOM_MODE.STANDBY AND NOT GVL.RM44_3_DEPROX_SWITCH);
(* ROOMT STATUS *)
FB_ROOM_STATE_0(DEPROX_SWITCH := GVL.RM44_3_DEPROX_SWITCH, MODE_SWITCH := RM_MODE, IS_ALARM := GVL.RM44_3_InAlarm);
GVL.RM44_3_STATE := FB_ROOM_STATE_0.OUTPUT;
END_PROGRAM

PROGRAM RM51_STATUS
  VAR
    RM_MODE : ET_ROOM_MODE;
    ALARM_DELAY : TON;
    IS_ALARM : BOOL;
    TOF_BUZZER : TOF;
    RM_BUZZER_LOCAL : BOOL;
    IS_LOCAL_ALARM : BOOL;
    FB_ROOM_STATE_0 : FB_ROOM_STATE;
  END_VAR

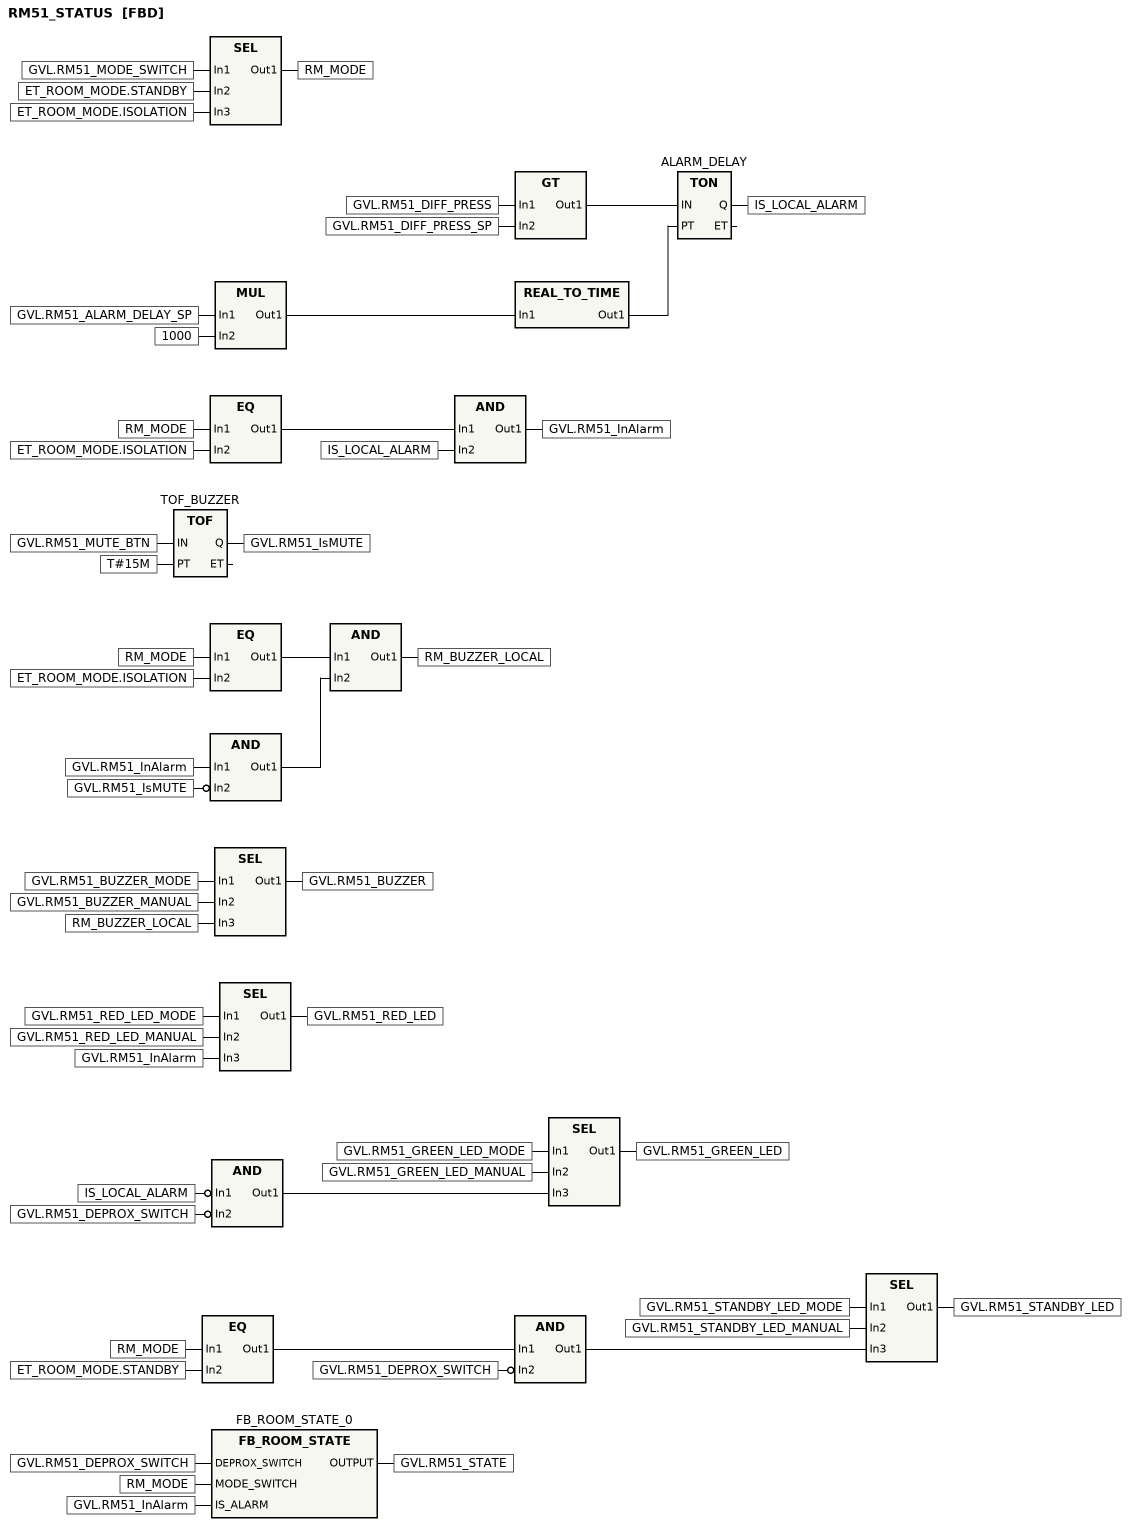
(* FBD diagram, written out as Structured Text *)
(* The mode switch located on the room alarm panel is to switch the room status between isolation mode and standby mode. *)
RM_MODE := SEL(GVL.RM51_MODE_SWITCH, ET_ROOM_MODE.STANDBY, ET_ROOM_MODE.ISOLATION);
(* generate alarms when RM DIFF PRESS >  RM DIFF PRESS SP.
the alarm will show on LED *)
ALARM_DELAY(IN := GVL.RM51_DIFF_PRESS > GVL.RM51_DIFF_PRESS_SP, PT := REAL_TO_TIME(GVL.RM51_ALARM_DELAY_SP * 1000));
IS_LOCAL_ALARM := ALARM_DELAY.Q;
(* ROOM IN ALARM *)
GVL.RM51_InAlarm := RM_MODE = ET_ROOM_MODE.ISOLATION AND IS_LOCAL_ALARM;
(* BUZZER
If the room is operating in isolation mode, the buzzer will activate until the panel RED button is pressed by an operator. If the room pressure remains outside of the acceptable range for a further 15 minutes, then the room buzzer will re-enable.

DISABLE BUZZER *)
TOF_BUZZER(IN := GVL.RM51_MUTE_BTN, PT := T#15M);
GVL.RM51_IsMUTE := TOF_BUZZER.Q;
(* BUZZER
If the room is operating in isolation mode, the buzzer will activate until the panel RED button is pressed by an operator. If the room pressure remains outside of the acceptable range for a further 15 minutes, then the room buzzer will re-enable. *)
RM_BUZZER_LOCAL := RM_MODE = ET_ROOM_MODE.ISOLATION AND GVL.RM51_InAlarm AND NOT GVL.RM51_IsMUTE;
(* AUTO/ MANUAL  MODE FROM BMS / BUZZER *)
GVL.RM51_BUZZER := SEL(GVL.RM51_BUZZER_MODE, GVL.RM51_BUZZER_MANUAL, RM_BUZZER_LOCAL);
(* AUTO/ MANUAL  MODE FROM BMS / RED LED *)
GVL.RM51_RED_LED := SEL(GVL.RM51_RED_LED_MODE, GVL.RM51_RED_LED_MANUAL, GVL.RM51_InAlarm);
(* AUTO/ MANUAL  MODE FROM BMS / GREEN LED *)
GVL.RM51_GREEN_LED := SEL(GVL.RM51_GREEN_LED_MODE, GVL.RM51_GREEN_LED_MANUAL, NOT IS_LOCAL_ALARM AND NOT GVL.RM51_DEPROX_SWITCH);
GVL.RM51_STANDBY_LED := SEL(GVL.RM51_STANDBY_LED_MODE, GVL.RM51_STANDBY_LED_MANUAL, RM_MODE = ET_ROOM_MODE.STANDBY AND NOT GVL.RM51_DEPROX_SWITCH);
(* ROOMT STATUS *)
FB_ROOM_STATE_0(DEPROX_SWITCH := GVL.RM51_DEPROX_SWITCH, MODE_SWITCH := RM_MODE, IS_ALARM := GVL.RM51_InAlarm);
GVL.RM51_STATE := FB_ROOM_STATE_0.OUTPUT;
END_PROGRAM

PROGRAM RM53_STATUS
  VAR
    RM_MODE : ET_ROOM_MODE;
    ALARM_DELAY : TON;
    IS_ALARM : BOOL;
    TOF_BUZZER : TOF;
    RM_BUZZER_LOCAL : BOOL;
    IS_LOCAL_ALARM : BOOL;
    FB_ROOM_STATE_0 : FB_ROOM_STATE;
  END_VAR

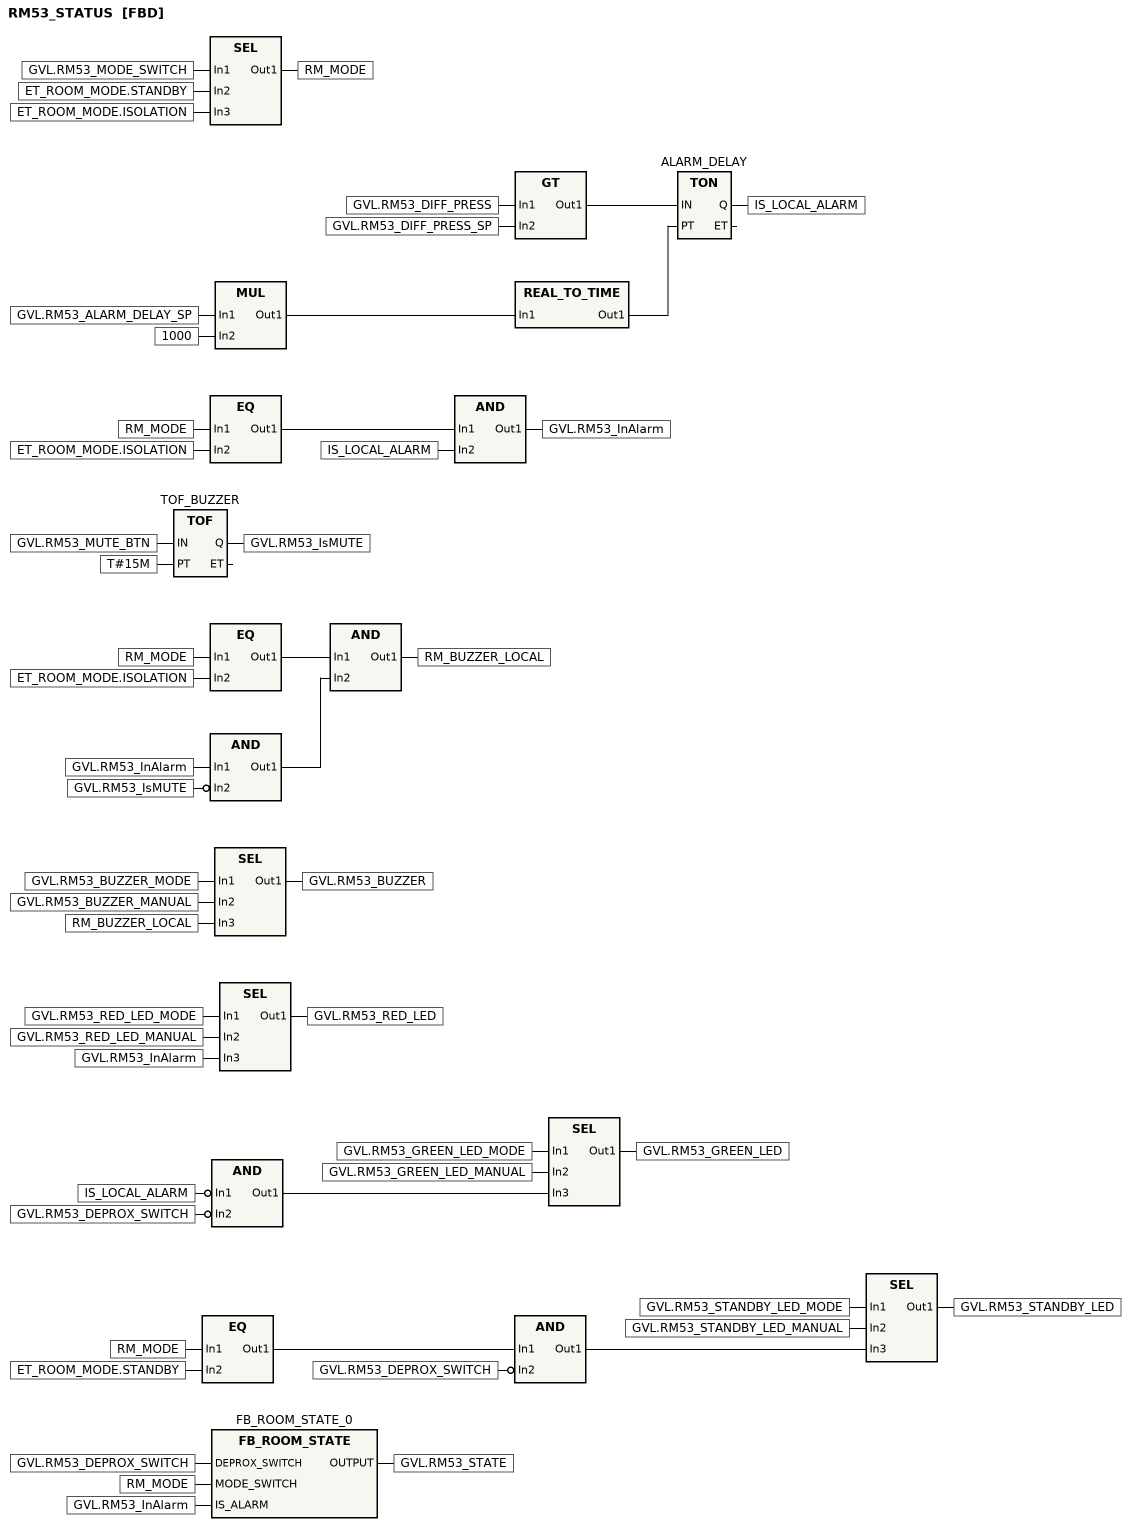
(* FBD diagram, written out as Structured Text *)
(* The mode switch located on the room alarm panel is to switch the room status between isolation mode and standby mode. *)
RM_MODE := SEL(GVL.RM53_MODE_SWITCH, ET_ROOM_MODE.STANDBY, ET_ROOM_MODE.ISOLATION);
(* generate alarms when RM DIFF PRESS >  RM DIFF PRESS SP.
the alarm will show on LED *)
ALARM_DELAY(IN := GVL.RM53_DIFF_PRESS > GVL.RM53_DIFF_PRESS_SP, PT := REAL_TO_TIME(GVL.RM53_ALARM_DELAY_SP * 1000));
IS_LOCAL_ALARM := ALARM_DELAY.Q;
(* ROOM IN ALARM *)
GVL.RM53_InAlarm := RM_MODE = ET_ROOM_MODE.ISOLATION AND IS_LOCAL_ALARM;
(* BUZZER
If the room is operating in isolation mode, the buzzer will activate until the panel RED button is pressed by an operator. If the room pressure remains outside of the acceptable range for a further 15 minutes, then the room buzzer will re-enable.

DISABLE BUZZER *)
TOF_BUZZER(IN := GVL.RM53_MUTE_BTN, PT := T#15M);
GVL.RM53_IsMUTE := TOF_BUZZER.Q;
(* BUZZER
If the room is operating in isolation mode, the buzzer will activate until the panel RED button is pressed by an operator. If the room pressure remains outside of the acceptable range for a further 15 minutes, then the room buzzer will re-enable. *)
RM_BUZZER_LOCAL := RM_MODE = ET_ROOM_MODE.ISOLATION AND GVL.RM53_InAlarm AND NOT GVL.RM53_IsMUTE;
(* AUTO/ MANUAL  MODE FROM BMS / BUZZER *)
GVL.RM53_BUZZER := SEL(GVL.RM53_BUZZER_MODE, GVL.RM53_BUZZER_MANUAL, RM_BUZZER_LOCAL);
(* AUTO/ MANUAL  MODE FROM BMS / RED LED *)
GVL.RM53_RED_LED := SEL(GVL.RM53_RED_LED_MODE, GVL.RM53_RED_LED_MANUAL, GVL.RM53_InAlarm);
(* AUTO/ MANUAL  MODE FROM BMS / GREEN LED *)
GVL.RM53_GREEN_LED := SEL(GVL.RM53_GREEN_LED_MODE, GVL.RM53_GREEN_LED_MANUAL, NOT IS_LOCAL_ALARM AND NOT GVL.RM53_DEPROX_SWITCH);
GVL.RM53_STANDBY_LED := SEL(GVL.RM53_STANDBY_LED_MODE, GVL.RM53_STANDBY_LED_MANUAL, RM_MODE = ET_ROOM_MODE.STANDBY AND NOT GVL.RM53_DEPROX_SWITCH);
(* ROOMT STATUS *)
FB_ROOM_STATE_0(DEPROX_SWITCH := GVL.RM53_DEPROX_SWITCH, MODE_SWITCH := RM_MODE, IS_ALARM := GVL.RM53_InAlarm);
GVL.RM53_STATE := FB_ROOM_STATE_0.OUTPUT;
END_PROGRAM

FUNCTION_BLOCK FB_PULSE_GENERATOR
  VAR_INPUT
    ENABLE : BOOL;
  END_VAR
  VAR_OUTPUT
    OUTPUT : BOOL;
  END_VAR
  VAR
    PULSESTATE : BOOL;
    PULSETIME : INT;
  END_VAR

                    
IF (ENABLE) THEN
	IF(PULSETIME > 100) THEN
		PULSESTATE := NOT PULSESTATE;
		PULSETIME := 0;
	END_IF;
	IF (PULSETIME < 0) THEN
		PULSETIME := 0;
	END_IF;
ELSE
	PULSESTATE := FALSE;
	PULSETIME := 0;
END_IF;

PULSETIME := PULSETIME +1;

OUTPUT := PULSESTATE;
                  
END_FUNCTION_BLOCK

PROGRAM RM44_3_DEPROX
  VAR
    ENABLE_BLINKING : BOOL;
    FB_PULSE_GENERATOR_0 : FB_PULSE_GENERATOR;
  END_VAR

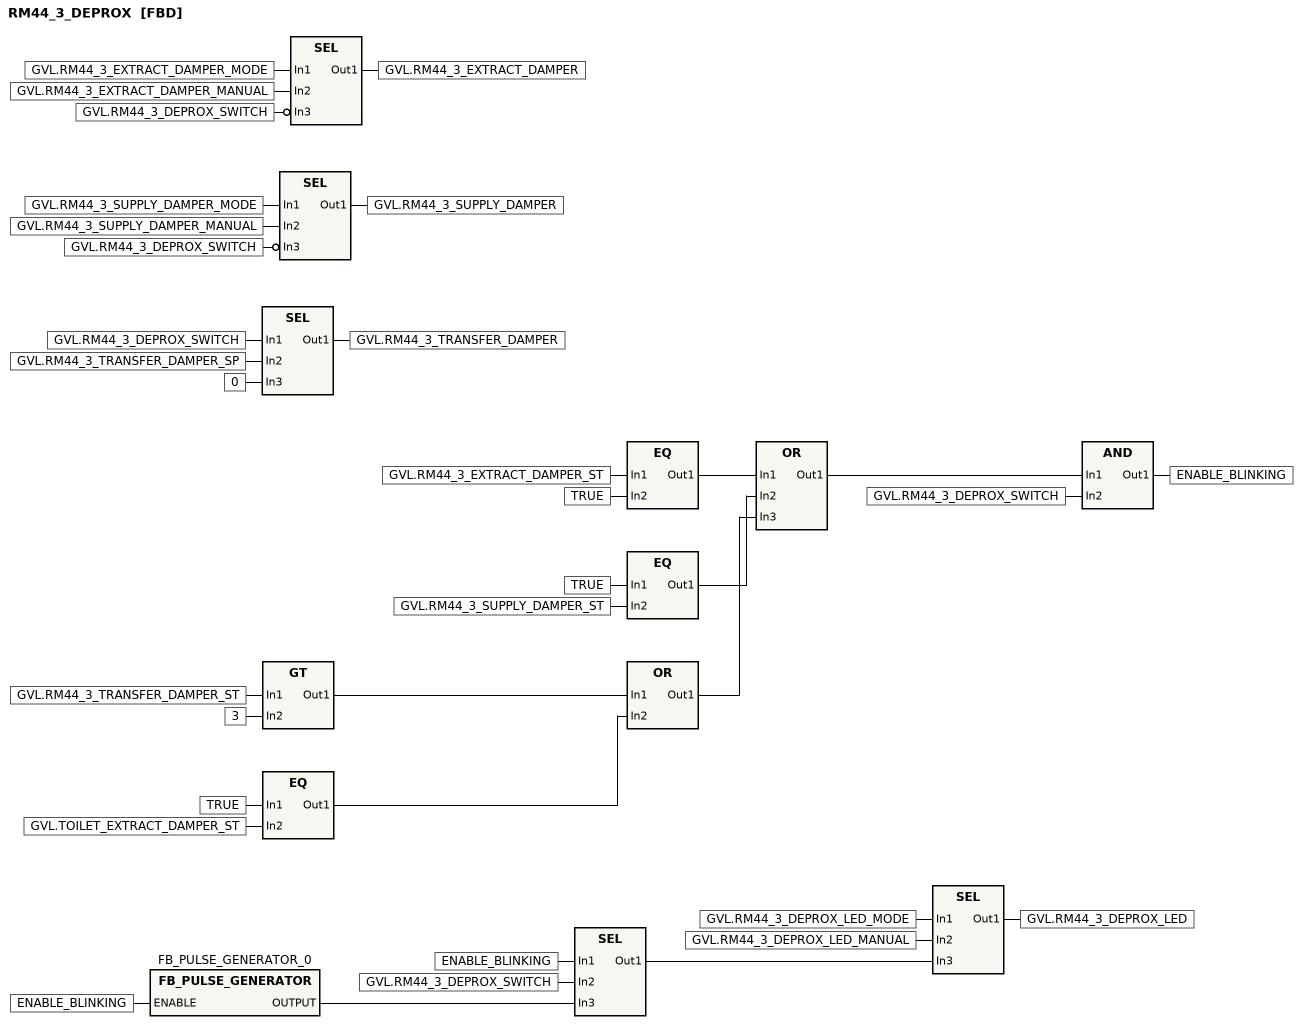
(* FBD diagram, written out as Structured Text *)
(* Return Air Damper - close damper in deprox mode

Deprox Switch. 0=normal 1=deprox *)
GVL.RM44_3_EXTRACT_DAMPER := SEL(GVL.RM44_3_EXTRACT_DAMPER_MODE, GVL.RM44_3_EXTRACT_DAMPER_MANUAL, NOT GVL.RM44_3_DEPROX_SWITCH);
(* Supply Air Damper - close damper in deprox mode

Deprox Switch. 0=normal 1=deprox *)
GVL.RM44_3_SUPPLY_DAMPER := SEL(GVL.RM44_3_SUPPLY_DAMPER_MODE, GVL.RM44_3_SUPPLY_DAMPER_MANUAL, NOT GVL.RM44_3_DEPROX_SWITCH);
(* Transfer Damper - close damper in deprox mode

Deprox Switch. 0=normal 1=deprox *)
GVL.RM44_3_TRANSFER_DAMPER := SEL(GVL.RM44_3_DEPROX_SWITCH, GVL.RM44_3_TRANSFER_DAMPER_SP, 0);
(* enable blinking when the room dampers are driving closed *)
ENABLE_BLINKING := (GVL.RM44_3_EXTRACT_DAMPER_ST = TRUE OR TRUE = GVL.RM44_3_SUPPLY_DAMPER_ST OR GVL.RM44_3_TRANSFER_DAMPER_ST > 3 OR TRUE = GVL.TOILET_EXTRACT_DAMPER_ST) AND GVL.RM44_3_DEPROX_SWITCH;
(* DEPROX LED *)
FB_PULSE_GENERATOR_0(ENABLE := ENABLE_BLINKING);
GVL.RM44_3_DEPROX_LED := SEL(GVL.RM44_3_DEPROX_LED_MODE, GVL.RM44_3_DEPROX_LED_MANUAL, SEL(ENABLE_BLINKING, GVL.RM44_3_DEPROX_SWITCH, FB_PULSE_GENERATOR_0.OUTPUT));
END_PROGRAM

FUNCTION_BLOCK FB_ROOM_STATE
  VAR_INPUT
    DEPROX_SWITCH : BOOL;
    MODE_SWITCH : ET_ROOM_MODE;
    IS_ALARM : BOOL;
  END_VAR
  VAR_OUTPUT
    OUTPUT : ET_ROOM_STATE;
  END_VAR

                    IF (DEPROX_SWITCH) THEN
	OUTPUT:= ET_ROOM_STATE.DEPROX;
ELSIF (MODE_SWITCH = ET_ROOM_MODE.STANDBY) THEN
	OUTPUT := ET_ROOM_STATE.STANDBY;
ELSIF ((MODE_SWITCH = ET_ROOM_MODE.ISOLATION) AND IS_ALARM) THEN
	OUTPUT := ET_ROOM_STATE.ALARM;
ELSE
	OUTPUT := ET_ROOM_STATE.ISOLATE;
END_IF;
                  
END_FUNCTION_BLOCK

PROGRAM RM59_DEPROX
  VAR
    ENABLE_BLINKING : BOOL;
    FB_PULSE_GENERATOR_0 : FB_PULSE_GENERATOR;
  END_VAR

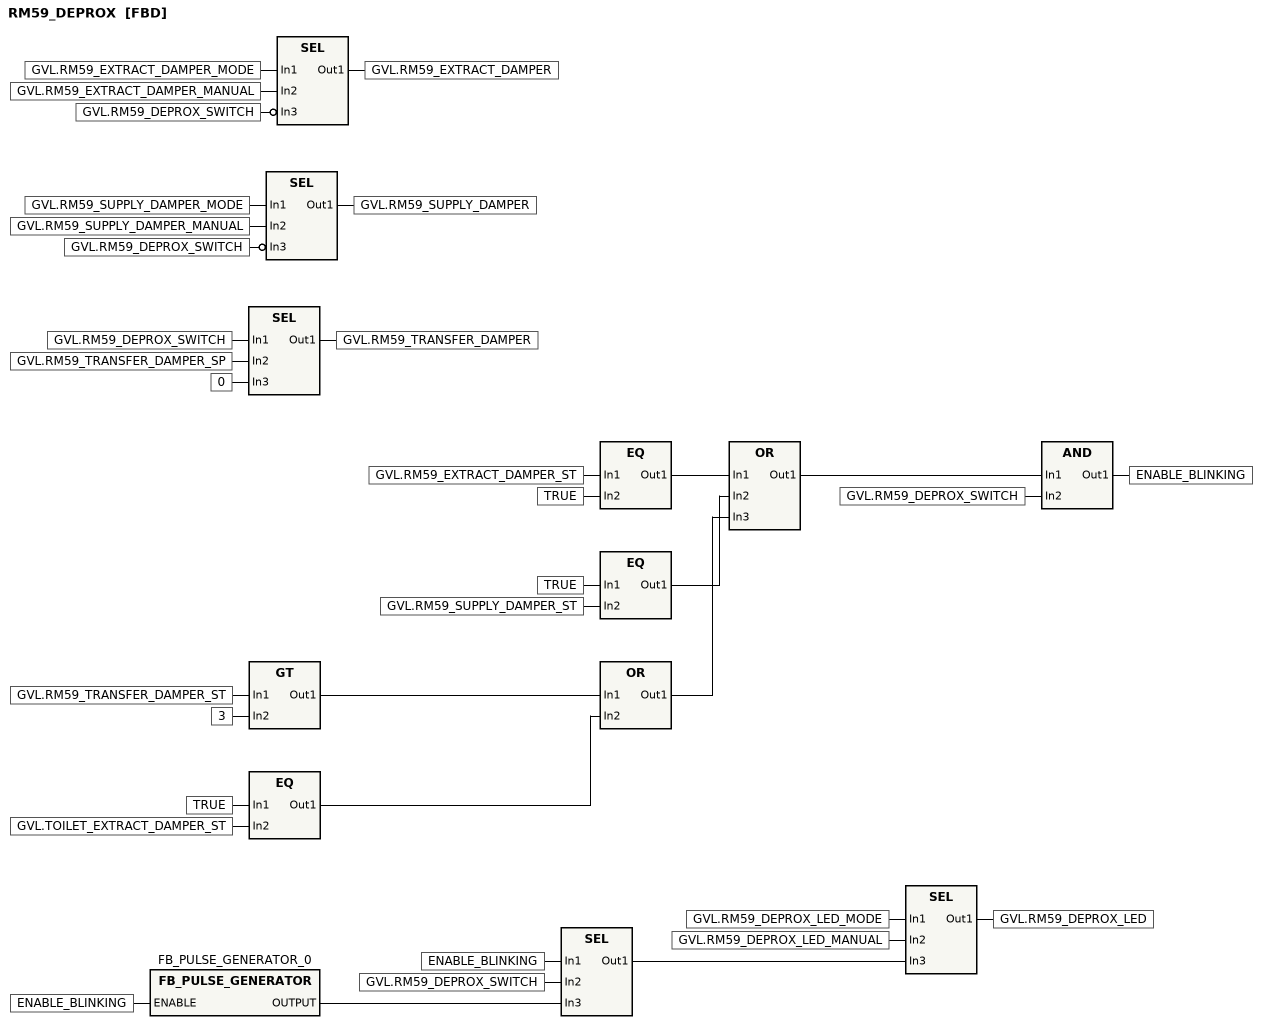
(* FBD diagram, written out as Structured Text *)
(* Return Air Damper - close damper in deprox mode

Deprox Switch. 0=normal 1=deprox *)
GVL.RM59_EXTRACT_DAMPER := SEL(GVL.RM59_EXTRACT_DAMPER_MODE, GVL.RM59_EXTRACT_DAMPER_MANUAL, NOT GVL.RM59_DEPROX_SWITCH);
(* Supply Air Damper - close damper in deprox mode

Deprox Switch. 0=normal 1=deprox *)
GVL.RM59_SUPPLY_DAMPER := SEL(GVL.RM59_SUPPLY_DAMPER_MODE, GVL.RM59_SUPPLY_DAMPER_MANUAL, NOT GVL.RM59_DEPROX_SWITCH);
(* Transfer Damper - close damper in deprox mode

Deprox Switch. 0=normal 1=deprox *)
GVL.RM59_TRANSFER_DAMPER := SEL(GVL.RM59_DEPROX_SWITCH, GVL.RM59_TRANSFER_DAMPER_SP, 0);
(* enable blinking when the room dampers are driving closed *)
ENABLE_BLINKING := (GVL.RM59_EXTRACT_DAMPER_ST = TRUE OR TRUE = GVL.RM59_SUPPLY_DAMPER_ST OR GVL.RM59_TRANSFER_DAMPER_ST > 3 OR TRUE = GVL.TOILET_EXTRACT_DAMPER_ST) AND GVL.RM59_DEPROX_SWITCH;
(* DEPROX LED *)
FB_PULSE_GENERATOR_0(ENABLE := ENABLE_BLINKING);
GVL.RM59_DEPROX_LED := SEL(GVL.RM59_DEPROX_LED_MODE, GVL.RM59_DEPROX_LED_MANUAL, SEL(ENABLE_BLINKING, GVL.RM59_DEPROX_SWITCH, FB_PULSE_GENERATOR_0.OUTPUT));
END_PROGRAM

FUNCTION_BLOCK FB_TOTAL_DEPROX
  VAR_OUTPUT
    DEPROX_ENABLE : BOOL;
    DEPROX_1RM : BOOL;
    DEPROX_2RM : BOOL;
  END_VAR
  VAR
    countRoom : INT := 0;
  END_VAR
  VAR_INPUT
    isRM1_DEPROX : BOOL;
    isRM2_DEPROX : BOOL;
    isRM3_DEPROX : BOOL;
    isRM4_DEPROX : BOOL;
    isRM5_DEPROX : BOOL;
    isRM6_DEPROX : BOOL;
    isRM7_DEPROX : BOOL;
    isRM8_DEPROX : BOOL;
    isRM9_DEPROX : BOOL;
    isRM10_DEPROX : BOOL;
  END_VAR

                    countRoom :=0;

IF (isRM1_DEPROX) THEN
	countRoom := countRoom + 1;
END_IF;

IF (isRM2_DEPROX) THEN
	countRoom := countRoom + 1;
END_IF;

IF (isRM3_DEPROX) THEN
	countRoom := countRoom + 1;
END_IF;

IF (isRM4_DEPROX) THEN
	countRoom := countRoom + 1;
END_IF;

IF (isRM5_DEPROX) THEN
	countRoom := countRoom + 1;
END_IF;

IF (isRM6_DEPROX) THEN
	countRoom := countRoom + 1;
END_IF;

IF (isRM7_DEPROX) THEN
	countRoom := countRoom + 1;
END_IF;

IF (isRM8_DEPROX) THEN
	countRoom := countRoom + 1;
END_IF;

IF (isRM9_DEPROX) THEN
	countRoom := countRoom + 1;
END_IF;

IF (isRM10_DEPROX) THEN
	countRoom := countRoom + 1;
END_IF;

IF (countRoom = 0) THEN 
	DEPROX_ENABLE := FALSE;
	DEPROX_1RM := FALSE;
	DEPROX_2RM := FALSE;
ELSIF (countRoom = 1) THEN 
	DEPROX_ENABLE := TRUE;
	DEPROX_1RM := TRUE;
	DEPROX_2RM := FALSE;
ELSIF (countRoom = 2) THEN 
	DEPROX_ENABLE := TRUE;
	DEPROX_1RM := TRUE;
	DEPROX_2RM := FALSE;
ELSIF (countRoom = 3) THEN 
	DEPROX_ENABLE := TRUE;
	DEPROX_1RM := TRUE;
	DEPROX_2RM := FALSE;
ELSE
	DEPROX_ENABLE := TRUE;
	DEPROX_1RM := FALSE;
	DEPROX_2RM := TRUE;
END_IF
                  
END_FUNCTION_BLOCK

(* Implicitly generated code : DO NOT EDIT *)
{attribute 'check_bounds'}
{attribute 'no_check'}
FUNCTION CheckBounds : DINT
  VAR_INPUT
    index : DINT;
    lower : DINT;
    upper : DINT;
  END_VAR

                    // Implicitly generated code : Only an Implementation suggestion
IF  index < lower THEN
	CheckBounds := lower;
ELSIF  index > upper THEN
	CheckBounds := upper;
ELSE  
	CheckBounds := index;
END_IF

(*It is also possible to set a breakpoint, log messages or e.g. to halt on an exception:
Add CmpApp.library, SysExcept.library and SysTypes2_Itf as newest.
Declaration:
VAR
    _pApp : POINTER TO CmpApp.APPLICATION;
    _result   : SysTypes.RTS_IEC_RESULT;
END_VAR

Implementation:
_pApp := AppGetCurrent(pResult:=_result);
IF  index < lower THEN
        CheckBounds := lower;
        IF _pApp <> 0 THEN
                AppGenerateException(pApp:=_pApp, ulException:=RtsExceptions.RTSEXCPT_ARRAYBOUNDS);
        END_IF
ELSIF  index > upper THEN
        CheckBounds := upper;
        IF _pApp <> 0 THEN
                AppGenerateException(pApp:=_pApp,   ulException:=RtsExceptions.RTSEXCPT_ARRAYBOUNDS);
        END_IF
ELSE  
        CheckBounds := index;
END_IF
*)

                  
END_FUNCTION

FUNCTION_BLOCK FB_9StatesMonitoring
  VAR
    ENABLE_OFF : BOOL := FALSE;
    ENABLE_ON : BOOL := FALSE;
    STATUS_ON : BOOL := FALSE;
    STATUS_OFF : BOOL := FALSE;
    FIRE_ON : BOOL := FALSE;
    FIRE_OFF : BOOL := FALSE;
    BEEN_RUNNING_OK : BOOL := FALSE;
    NOT_BEEN_RUNNING_OK : BOOL := FALSE;
    ALL_OFF : BOOL := FALSE;
    NOT_ALL_OFF : BOOL := FALSE;
    START_DELAY_ON : BOOL := FALSE;
    START_DELAY_OFF : BOOL := FALSE;
    STOP_DELAY_ON : BOOL := FALSE;
    STOP_DELAY_OFF : BOOL := FALSE;
    ENABLE_TIMER_ON : BOOL := FALSE;
    ENABLE_TIMER_OFF : BOOL := FALSE;
    BEEN_RUNNING_OK_LATCH : RS;
    ALL_OFF_LATCH : RS;
    START_DELAY_TON : TON;
    STOP_DELAY_TON : TON;
    STOPPED : INT;
  END_VAR
  VAR_INPUT
    ENABLE : BOOL := FALSE;
    STATUS : BOOL := FALSE;
    FIRE : BOOL := FALSE;
  END_VAR
  VAR_OUTPUT
    STATE : ET_9STATE_MONITORING := 9;
  END_VAR

                    (* 
Version 1.0
Last Updated: 28/01/2020

9 States Monitoring. Value from 0 to 9
	STOPPED := 0,
	RUNNING := 1,
	STARTING := 2,
	STOPPING := 3,
	START_FAIL := 4,
	STOP_FAIL := 5,
	UNEXPECTED_START := 6,
	UNEXPECTED_STOP := 7,
	FIRE_STOP := 8,
	UNKNOWN := 9
*)

ENABLE_OFF := (ENABLE = FALSE);
ENABLE_ON := (ENABLE = TRUE);
STATUS_ON := (STATUS = TRUE);
STATUS_OFF := (STATUS = FALSE);
FIRE_ON := (FIRE = TRUE);
FIRE_OFF := (FIRE = FALSE);

BEEN_RUNNING_OK_LATCH(SET := ENABLE_ON AND STATUS_ON, RESET1 := ENABLE_OFF);
BEEN_RUNNING_OK := BEEN_RUNNING_OK_LATCH.Q1;

ALL_OFF_LATCH(SET := ENABLE_OFF AND STATUS_OFF, RESET1 := ENABLE_ON);
ALL_OFF := ALL_OFF_LATCH.Q1;

START_DELAY_TON(IN := ENABLE_ON, PT := T#30S);
START_DELAY_ON := START_DELAY_TON.Q;

STOP_DELAY_TON(IN := ENABLE_OFF, PT := T#30S);
STOP_DELAY_ON := STOP_DELAY_TON.Q;

ENABLE_TIMER_ON := ((START_DELAY_TON.ET < T#30S AND ENABLE_ON) OR (STOP_DELAY_TON.ET < T#30S AND ENABLE_OFF));

START_DELAY_OFF := NOT START_DELAY_ON;
STOP_DELAY_OFF := NOT STOP_DELAY_ON;
ENABLE_TIMER_OFF := NOT ENABLE_TIMER_ON;
NOT_BEEN_RUNNING_OK := NOT BEEN_RUNNING_OK;
NOT_ALL_OFF := NOT ALL_OFF;

IF (ENABLE_ON AND STATUS_OFF AND FIRE_ON) THEN
	STATE := ET_9STATE_MONITORING.FIRE_STOP;
ELSIF (ENABLE_OFF AND STATUS_ON AND STOP_DELAY_ON AND NOT_BEEN_RUNNING_OK AND NOT_ALL_OFF) THEN
	STATE := ET_9STATE_MONITORING.STOP_FAIL;
ELSIF (ENABLE_ON AND STATUS_OFF AND START_DELAY_ON AND NOT_BEEN_RUNNING_OK AND NOT_ALL_OFF) THEN
	STATE := ET_9STATE_MONITORING.START_FAIL;
ELSIF (ENABLE_OFF AND STATUS_ON AND ENABLE_TIMER_OFF AND STOP_DELAY_ON AND ENABLE_TIMER_OFF AND ALL_OFF) THEN
	STATE := ET_9STATE_MONITORING.UNEXPECTED_START;
ELSIF (ENABLE_ON AND STATUS_OFF AND START_DELAY_ON AND FIRE_OFF AND ENABLE_TIMER_OFF AND BEEN_RUNNING_OK AND NOT_ALL_OFF) THEN
	STATE := ET_9STATE_MONITORING.UNEXPECTED_STOP;
ELSIF (ENABLE_OFF AND STATUS_ON AND ENABLE_TIMER_ON AND STOP_DELAY_OFF AND FIRE_OFF) THEN
	STATE := ET_9STATE_MONITORING.STOPPING;
ELSIF (ENABLE_ON AND STATUS_ON) THEN
	STATE := ET_9STATE_MONITORING.RUNNING;
ELSIF (ENABLE_ON AND STATUS_OFF AND ENABLE_TIMER_ON AND START_DELAY_OFF AND FIRE_OFF) THEN
	STATE := ET_9STATE_MONITORING.STARTING;
ELSIF (ENABLE_OFF AND STATUS_OFF) THEN
	STATE := ET_9STATE_MONITORING.STOPPED;
ELSE
	STATE := ET_9STATE_MONITORING.UNKNOWN;
END_IF;
                  
END_FUNCTION_BLOCK

FUNCTION_BLOCK FB_2_10V_TO_0_10V_INPUT
  VAR_INPUT
    IN_PRCT : REAL;  (* 0-10V = 0-100% *)
  END_VAR
  VAR_OUTPUT
    OUT_PRCT : REAL;  (* 2-10V = 0-100% *)
  END_VAR
  VAR
    result : REAL;
    LIN : FB_LINEAR;
  END_VAR

                    LIN (X1:=2, Y1:=0, X2:=10, Y2:=10, INPUT:= IN_PRCT/10);
OUT_PRCT := MAX(0, MIN(LIN.OUTPUT * 10, 100));

                  
END_FUNCTION_BLOCK

PROGRAM DEPROX_SIGNAL

                    IF(GVL.RM71_DEPROX_SWITCH AND GVL.RM74_DEPROX_SWITCH ) THEN 
	GVL.DEPROX_SIGNAL1 := TRUE;
	GVL.DEPROX_SIGNAL2 := TRUE;
ELSIF(GVL.RM71_DEPROX_SWITCH OR GVL.RM74_DEPROX_SWITCH) THEN
	GVL.DEPROX_SIGNAL1 := TRUE;
	GVL.DEPROX_SIGNAL2 := FALSE;
ELSE
	GVL.DEPROX_SIGNAL1 := FALSE;
	GVL.DEPROX_SIGNAL2 := FALSE;
END_IF;
                  
END_PROGRAM

FUNCTION_BLOCK FB_LINEAR
  VAR_INPUT
    X1 : REAL;
    Y1 : REAL;
    X2 : REAL;
    Y2 : REAL;
    INPUT : REAL;
  END_VAR
  VAR
    m : REAL;
  END_VAR
  VAR_OUTPUT
    OUTPUT : REAL;
  END_VAR

                    // (y-y1) = m(x-x1)
// m = (y2-y1)/(x2-x1)

m := (Y2-Y1) / (X2-X1);
OUTPUT := (m * (INPUT-X1)) + Y1;
                  
END_FUNCTION_BLOCK

PROGRAM OUTPUT_MAPPING
  VAR
    voltage_converter : FB_0_10V_TO_2_10V_OUTPUT;
  END_VAR

                    //MODULE 1
voltage_converter(IN_PRCT := GVL.RM71_TRANSFER_DAMPER);
qRM71_TRANSFER_DAMPER := TRUNC_INT(120 - voltage_converter.OUT_PRCT) * 100; //AO0 0v=open 10v=close

voltage_converter(IN_PRCT := GVL.RM74_TRANSFER_DAMPER);
qRM74_TRANSFER_DAMPER := TRUNC_INT(120 - voltage_converter.OUT_PRCT) * 100; //AO1 0v=open 10v=close

//MODULE 2
voltage_converter(IN_PRCT := GVL.RM74_ADDITIONAL_TRANSFER_DAMPER);
qADDITIONAL_TRANSFER_DAMPER := TRUNC_INT(120 - voltage_converter.OUT_PRCT) * 100; //AO1 0v=open 10v=close

//MODULE 3
qRM71_RED_LED := GVL.RM71_RED_LED; //DO1
qRM71_GREEN_LED := GVL.RM71_GREEN_LED; //DO2
qRM71_STANDBY_LED := GVL.RM71_STANDBY_LED; //DO3
qRM71_DEPROX_LED := GVL.RM71_DEPROX_LED; //DO4
qRM71_BUZZER := GVL.RM71_BUZZER; //DO5
qRM74_RED_LED := GVL.RM74_RED_LED; //DO6
qRM74_GREEN_LED := GVL.RM74_GREEN_LED; //DO7
qRM74_STANDBY_LED := GVL.RM74_STANDBY_LED; //DO8
qRM74_DEPROX_LED := GVL.RM74_DEPROX_LED; //DO9
qRM74_BUZZER := GVL.RM74_BUZZER; //DO10

//MODULE 4
qRM71_SUPPLY_DAMPER_POS := NOT GVL.RM71_SUPPLY_DAMPER;  //DO1
qRM74_SUPPLY_DAMPER_POS  := NOT GVL.RM74_SUPPLY_DAMPER ; //DO2
qRM71_EXHAUST_DAMPER_POS  := NOT GVL.RM71_EXTRACT_DAMPER ; //DO3
qRM74_EXHAUST_DAMPER_POS  := NOT  GVL.RM74_EXTRACT_DAMPER ; //DO4
qDEPROX_SIGNAL1 := GVl.DEPROX_SIGNAL1; //DO5 // 1 ROOM  in deprox mode
qDEPROX_SIGNAL2 := GVl.DEPROX_SIGNAL2; //DO6 // 2 rooms in deprox mode

                  
END_PROGRAM

PROGRAM INPUT_MAPPING
  VAR
    voltage_converter : FB_2_10V_TO_0_10V_INPUT;
    VPRaw : REAL;
    voltage_converter1 : FB_2_10V_TO_0_10V_INPUT;
  END_VAR

                    (*
	2 Rooms - Buzzer, Green LED and Red LED for each room
	
	check MAST to see which programs get execture

*)


voltage_converter1(IN_PRCT := INT_TO_REAL(iRM71_TRANSFER_DAMPER_ST));
GVL.RM71_TRANSFER_DAMPER_ST := 100 - voltage_converter1.OUT_PRCT; //AI0  0v=open 10v=close

voltage_converter(IN_PRCT := INT_TO_REAL(iRM74_TRANSFER_DAMPER_ST));
GVL.RM74_TRANSFER_DAMPER_ST := 100 - voltage_converter.OUT_PRCT; //AI1  0v=open 10v=close

GVL.RM71_HALL_TO_RM_DIFF_PRESS  := INT_TO_REAL(iRM71_HALL_TO_RM_DIFF_PRESS); //AI2
GVL.RM71_ANTE_TO_RM_DIFF_PRESS  := INT_TO_REAL(iRM71_ANTE_TO_RM_DIFF_PRESS); //AI3

//MODULE 2
GVL.RM71_HALL_TO_ANTE_DIFF_PRESS  := INT_TO_REAL(iRM71_HALL_TO_ANTE_DIFF_PRESS); //AI1
GVL.RM74_HALL_TO_RM_DIFF_PRESS  := INT_TO_REAL(iRM74_HALL_TO_RM_DIFF_PRESS); //AI2
GVL.RM74_ANTEL_TO_RM_DIFF_PRESS  := INT_TO_REAL(iRM74_ANTEL_TO_RM_DIFF_PRESS); //AI3
GVL.RM74_HALL_TO_ANTE_DIFF_PRESS  := INT_TO_REAL(iRM74_HALL_TO_ANTE_DIFF_PRESS); //AI4

//MODULE 4
GVL.RM71_SUPPLY_DAMPER_ST := NOT iRM71_SUPPLY_DAMPER_ST; //DI1
GVL.RM74_SUPPLY_DAMPER_ST :=  iRM74_SUPPLY_DAMPER_ST; //DI2
GVL.RM71_EXTRACT_DAMPER_ST := NOT iRM71_EXTRACT_DAMPER_ST; //DI3
GVL.RM74_EXTRACT_DAMPER_ST :=  iRM74_EXTRACT_DAMPER_ST; //DI4
GVL.RM71_MODE_SWITCH := iRM71_NEGATIVE_MODE_SWITCH; //DI5
GVL.RM71_DEPROX_SWITCH := iRM71_DEPROX_SWITCH; //DI6
GVL.RM71_MUTE_BTN := iRM71_MUTE_BTN; //DI7
GVL.RM74_MODE_SWITCH := iRM74_NEGATIVE_MODE_SWITCH; //DI8
GVL.RM74_DEPROX_SWITCH := iRM74_DEPROX_SWITCH; //DI9
GVL.RM74_MUTE_BTN := iRM74_MUTE_BTN; //DI10

                  
END_PROGRAM

FUNCTION_BLOCK FB_ROOM_POSITIVE_STATE
  VAR_INPUT
    DEPROX_SWITCH : BOOL;
    MODE_SWITCH : ET_ROOM_MODE;
    IS_ALARM : BOOL;
  END_VAR
  VAR_OUTPUT
    OUTPUT : ET_ROOM_STATE;
  END_VAR
  VAR_INPUT
    POSITIVE_MODE : BOOL;
  END_VAR

                    IF (DEPROX_SWITCH) THEN
	OUTPUT:= ET_ROOM_STATE.DEPROX;
ELSIF (POSITIVE_MODE) THEN
	OUTPUT := ET_ROOM_STATE.POSITVE;
ELSIF (MODE_SWITCH = ET_ROOM_MODE.STANDBY) THEN
	OUTPUT := ET_ROOM_STATE.STANDBY;
ELSIF ((MODE_SWITCH = ET_ROOM_MODE.ISOLATION) AND IS_ALARM) THEN
	OUTPUT := ET_ROOM_STATE.ALARM;
ELSE
	OUTPUT := ET_ROOM_STATE.ISOLATE;
END_IF;
                  
END_FUNCTION_BLOCK

CONFIGURATION A02_CED_RESUS_ROOMS
  RESOURCE Application ON PLC
    VAR_GLOBAL  (* GVL *)
      RM6_DAMPER_POS : INT;
      RM9_DIFF_PRESS_NOTUSED : INT;
      RM119_DEPROX_SWITCH AT %MX2.3 : BOOL;  (* Input Mapping *)
      RM119_DEPROX_LED AT %MX2.0 : BOOL;  (* Output Mapping *)
      RM119_EXTRACT_DAMPER_ST AT %MX3.3 : BOOL;  (* Input Mapping *)
      RM119_EXTRACT_DAMPER AT %MX3.0 : BOOL;  (* Output Mapping *)
      RM119_SUPPLY_DAMPER_ST AT %MX8.3 : BOOL;  (* Input Mapping *)
      RM119_SUPPLY_DAMPER AT %MX8.0 : BOOL;  (* Output Mapping *)
      RM119_STATE AT %ML1501 : ET_ROOM_STATE;
      RM119_BUZZER AT %MX1.0 : BOOL;  (* output mapping *)
      RM119_DIFF_PRESS AT %MD501 : REAL;  (* Input Mapping *)
      RM119_InAlarm AT %MX5.0 : BOOL;
      RM119_IsMute AT %MX5.1 : BOOL;
      RM119_GREEN_LED AT %MX4.0 : BOOL;  (* OUTPUT_MAPPING *)
      RM119_MODE_SWITCH AT %MX5.2 : BOOL;  (* Input Mapping *)
      RM119_STANDBY_LED AT %MX7.0 : BOOL;  (* Output Mapping *)
      RM119_RED_LED AT %MX6.0 : BOOL;  (* Output Mapping *)
      RM119_MUTE_BTN AT %MX5.3 : BOOL;  (* Input Mapping *)
      RM119_TRANSFER_DAMPER AT %MD503 : REAL;  (* OUTPUT MAPPING *)
      RM119_TRANSFER_DAMPER_ST AT %MD505 : REAL;  (* INPUT MAPPING *)
      RM6_DEPROX_SWITCH AT %MX12.3 : BOOL;  (* Input Mapping *)
      RM6_DEPROX_LED AT %MX12.0 : BOOL;  (* Output Mapping *)
      RM6_EXTRACT_DAMPER1_ST AT %MD580 : REAL;  (* Input Mapping *)
      RM6_EXTRACT_DAMPER1 AT %MD578 : REAL;  (* Output Mapping *)
      RM6_SUPPLY_DAMPER_ST AT %MX18.3 : BOOL;  (* Input Mapping *)
      RM6_SUPPLY_DAMPER_NEG_SP AT %MD577 : REAL;
      RM6_SUPPLY_DAMPER_POS_SP AT %MD575 : REAL;
      RM6_SUPPLY_DAMPER AT %MD571 : REAL;  (* Output Mapping *)
      RM6_STATE AT %ML1502 : ET_ROOM_STATE;
      RM6_BUZZER AT %MX11.0 : BOOL;  (* output mapping *)
      RM6_DIFF_PRESS1 AT %MD506 : REAL;  (* Input Mapping *)
      RM6_InAlarm AT %MX15.0 : BOOL;
      RM6_IsMute AT %MX15.1 : BOOL;
      RM6_GREEN_LED AT %MX14.0 : BOOL;  (* OUTPUT_MAPPING *)
      RM6_MODE_SWITCH AT %MX15.2 : BOOL;  (* Input Mapping *)
      RM6_STANDBY_LED AT %MX17.0 : BOOL;  (* Output Mapping *)
      RM6_RED_LED AT %MX16.0 : BOOL;  (* Output Mapping *)
      RM6_MUTE_BTN AT %MX15.3 : BOOL;  (* Input Mapping *)
      RM6_TRANSFER_DAMPER AT %MD508 : REAL;  (* OUTPUT MAPPING *)
      RM6_TRANSFER_DAMPER_ST AT %MD510 : REAL;  (* INPUT MAPPING *)
      RM71_DEPROX_SWITCH AT %MX22.3 : BOOL;  (* Input Mapping *)
      RM71_DEPROX_LED AT %MX22.0 : BOOL;  (* Output Mapping *)
      RM71_EXTRACT_DAMPER_ST AT %MX23.3 : BOOL;  (* Input Mapping *)
      RM71_EXTRACT_DAMPER AT %MX23.0 : BOOL;  (* Output Mapping *)
      RM71_SUPPLY_DAMPER_ST AT %MX28.3 : BOOL;  (* Input Mapping *)
      RM71_SUPPLY_DAMPER AT %MX28.0 : BOOL;  (* Output Mapping *)
      RM71_STATE AT %ML1503 : ET_ROOM_STATE;
      RM71_BUZZER AT %MX21.0 : BOOL;  (* output mapping *)
      RM71_HALL_TO_RM_DIFF_PRESS AT %MD511 : REAL;  (* Input Mapping *)
      RM71_InAlarm AT %MX25.0 : BOOL;
      RM71_IsMute AT %MX25.1 : BOOL;
      RM71_GREEN_LED AT %MX24.0 : BOOL;  (* OUTPUT_MAPPING *)
      RM71_MODE_SWITCH AT %MX25.2 : BOOL;  (* Input Mapping *)
      RM71_STANDBY_LED AT %MX27.0 : BOOL;  (* Output Mapping *)
      RM71_RED_LED AT %MX26.0 : BOOL;  (* Output Mapping *)
      RM71_MUTE_BTN AT %MX25.3 : BOOL;  (* Input Mapping *)
      RM71_TRANSFER_DAMPER AT %MD513 : REAL;  (* OUTPUT MAPPING *)
      RM71_TRANSFER_DAMPER_ST AT %MD515 : REAL;  (* INPUT MAPPING *)
      RM74_DEPROX_SWITCH AT %MX32.3 : BOOL;  (* Input Mapping *)
      RM74_DEPROX_LED AT %MX32.0 : BOOL;  (* Output Mapping *)
      RM74_EXTRACT_DAMPER_ST AT %MX33.3 : BOOL;  (* Input Mapping *)
      RM74_EXTRACT_DAMPER AT %MX33.0 : BOOL;  (* Output Mapping *)
      RM74_SUPPLY_DAMPER_ST AT %MX38.3 : BOOL;  (* Input Mapping *)
      RM74_SUPPLY_DAMPER AT %MX38.0 : BOOL;  (* Output Mapping *)
      RM74_STATE AT %ML1504 : ET_ROOM_STATE;
      RM74_BUZZER AT %MX31.0 : BOOL;  (* output mapping *)
      RM74_HALL_TO_RM_DIFF_PRESS AT %MD516 : REAL;  (* Input Mapping *)
      RM74_InAlarm AT %MX35.0 : BOOL;
      RM74_IsMute AT %MX35.1 : BOOL;
      RM74_GREEN_LED AT %MX34.0 : BOOL;  (* OUTPUT_MAPPING *)
      RM74_MODE_SWITCH AT %MX35.2 : BOOL;  (* Input Mapping *)
      RM74_STANDBY_LED AT %MX37.0 : BOOL;  (* Output Mapping *)
      RM74_RED_LED AT %MX36.0 : BOOL;  (* Output Mapping *)
      RM74_MUTE_BTN AT %MX35.3 : BOOL;  (* Input Mapping *)
      RM74_TRANSFER_DAMPER AT %MD518 : REAL;  (* OUTPUT MAPPING *)
      RM74_TRANSFER_DAMPER_ST AT %MD520 : REAL;  (* INPUT MAPPING *)
      RM9_DEPROX_SWITCH AT %MX42.3 : BOOL;  (* Input Mapping *)
      RM9_DEPROX_LED AT %MX42.0 : BOOL;  (* Output Mapping *)
      RM9_EXTRACT_DAMPER_ST AT %MX43.3 : BOOL;  (* Input Mapping *)
      RM9_EXTRACT_DAMPER AT %MX43.0 : BOOL;  (* Output Mapping *)
      RM9_SUPPLY_DAMPER_ST AT %MX48.3 : BOOL;  (* Input Mapping *)
      RM9_SUPPLY_DAMPER AT %MX48.0 : BOOL;  (* Output Mapping *)
      RM9_STATE AT %ML1505 : ET_ROOM_STATE;
      RM9_BUZZER AT %MX41.0 : BOOL;  (* output mapping *)
      RM9_DIFF_PRESS1 AT %MD521 : REAL;  (* Input Mapping *)
      RM9_InAlarm AT %MX45.0 : BOOL;
      RM9_IsMute AT %MX45.1 : BOOL;
      RM9_GREEN_LED AT %MX44.0 : BOOL;  (* OUTPUT_MAPPING *)
      RM9_MODE_SWITCH AT %MX45.2 : BOOL;  (* Input Mapping *)
      RM9_STANDBY_LED AT %MX47.0 : BOOL;  (* Output Mapping *)
      RM9_RED_LED AT %MX46.0 : BOOL;  (* Output Mapping *)
      RM9_MUTE_BTN AT %MX45.3 : BOOL;  (* Input Mapping *)
      RM9_TRANSFER_DAMPER AT %MD523 : REAL;  (* OUTPUT MAPPING *)
      RM9_TRANSFER_DAMPER_ST AT %MD525 : REAL;  (* INPUT MAPPING *)
      RM44_3_DEPROX_SWITCH AT %MX52.3 : BOOL;  (* Input Mapping *)
      RM44_3_DEPROX_LED AT %MX52.0 : BOOL;  (* Output Mapping *)
      RM44_3_EXTRACT_DAMPER_ST AT %MX53.3 : BOOL;  (* Input Mapping *)
      RM44_3_EXTRACT_DAMPER AT %MX53.0 : BOOL;  (* Output Mapping *)
      RM44_3_SUPPLY_DAMPER_ST AT %MX58.3 : BOOL;  (* Input Mapping *)
      RM44_3_SUPPLY_DAMPER AT %MX58.0 : BOOL;  (* Output Mapping *)
      RM44_3_STATE AT %ML1506 : ET_ROOM_STATE;
      RM44_3_BUZZER AT %MX51.0 : BOOL;  (* output mapping *)
      RM44_3_DIFF_PRESS AT %MD526 : REAL;  (* Input Mapping *)
      RM44_3_InAlarm AT %MX55.0 : BOOL;
      RM44_3_IsMute AT %MX55.1 : BOOL;
      RM44_3_GREEN_LED AT %MX54.0 : BOOL;  (* OUTPUT_MAPPING *)
      RM44_3_MODE_SWITCH AT %MX55.2 : BOOL;  (* Input Mapping *)
      RM44_3_STANDBY_LED AT %MX57.0 : BOOL;  (* Output Mapping *)
      RM44_3_RED_LED AT %MX56.0 : BOOL;  (* Output Mapping *)
      RM44_3_MUTE_BTN AT %MX55.3 : BOOL;  (* Input Mapping *)
      RM44_3_TRANSFER_DAMPER AT %MD528 : REAL;  (* OUTPUT MAPPING *)
      RM44_3_TRANSFER_DAMPER_ST AT %MD530 : REAL;  (* INPUT MAPPING *)
      RM51_DEPROX_SWITCH AT %MX62.3 : BOOL;  (* Input Mapping *)
      RM51_DEPROX_LED AT %MX62.0 : BOOL;  (* Output Mapping *)
      RM51_EXTRACT_DAMPER_ST AT %MX63.3 : BOOL;  (* Input Mapping *)
      RM51_EXTRACT_DAMPER AT %MX63.0 : BOOL;  (* Output Mapping *)
      RM51_SUPPLY_DAMPER_ST AT %MX68.3 : BOOL;  (* Input Mapping *)
      RM51_SUPPLY_DAMPER AT %MX68.0 : BOOL;  (* Output Mapping *)
      RM51_STATE AT %ML1507 : ET_ROOM_STATE;
      RM51_BUZZER AT %MX61.0 : BOOL;  (* output mapping *)
      RM51_DIFF_PRESS AT %MD531 : REAL;  (* Input Mapping *)
      RM51_InAlarm AT %MX65.0 : BOOL;
      RM51_IsMute AT %MX65.1 : BOOL;
      RM51_GREEN_LED AT %MX64.0 : BOOL;  (* OUTPUT_MAPPING *)
      RM51_MODE_SWITCH AT %MX65.2 : BOOL;  (* Input Mapping *)
      RM51_STANDBY_LED AT %MX67.0 : BOOL;  (* Output Mapping *)
      RM51_RED_LED AT %MX66.0 : BOOL;  (* Output Mapping *)
      RM51_MUTE_BTN AT %MX65.3 : BOOL;  (* Input Mapping *)
      RM51_TRANSFER_DAMPER AT %MD533 : REAL;  (* OUTPUT MAPPING *)
      RM51_TRANSFER_DAMPER_ST AT %MD535 : REAL;  (* INPUT MAPPING *)
      RM52_DEPROX_SWITCH AT %MX72.3 : BOOL;  (* Input Mapping *)
      RM52_DEPROX_LED AT %MX72.0 : BOOL;  (* Output Mapping *)
      RM52_EXTRACT_DAMPER_ST AT %MX73.3 : BOOL;  (* Input Mapping *)
      RM52_EXTRACT_DAMPER AT %MX73.0 : BOOL;  (* Output Mapping *)
      RM52_SUPPLY_DAMPER_ST AT %MX78.3 : BOOL;  (* Input Mapping *)
      RM52_SUPPLY_DAMPER AT %MX78.0 : BOOL;  (* Output Mapping *)
      RM52_STATE AT %ML1508 : ET_ROOM_STATE;
      RM52_BUZZER AT %MX71.0 : BOOL;  (* output mapping *)
      RM52_DIFF_PRESS AT %MD536 : REAL;  (* Input Mapping *)
      RM52_InAlarm AT %MX75.0 : BOOL;
      RM52_IsMute AT %MX75.1 : BOOL;
      RM52_GREEN_LED AT %MX74.0 : BOOL;  (* OUTPUT_MAPPING *)
      RM52_MODE_SWITCH AT %MX75.2 : BOOL;  (* Input Mapping *)
      RM52_STANDBY_LED AT %MX77.0 : BOOL;  (* Output Mapping *)
      RM52_RED_LED AT %MX76.0 : BOOL;  (* Output Mapping *)
      RM52_MUTE_BTN AT %MX75.3 : BOOL;  (* Input Mapping *)
      RM52_TRANSFER_DAMPER AT %MD538 : REAL;  (* OUTPUT MAPPING *)
      RM52_TRANSFER_DAMPER_ST AT %MD540 : REAL;  (* INPUT MAPPING *)
      RM53_DEPROX_SWITCH AT %MX82.3 : BOOL;  (* Input Mapping *)
      RM53_DEPROX_LED AT %MX82.0 : BOOL;  (* Output Mapping *)
      RM53_EXTRACT_DAMPER_ST AT %MX83.3 : BOOL;  (* Input Mapping *)
      RM53_EXTRACT_DAMPER AT %MX83.0 : BOOL;  (* Output Mapping *)
      RM53_SUPPLY_DAMPER_ST AT %MX88.3 : BOOL;  (* Input Mapping *)
      RM53_SUPPLY_DAMPER AT %MX88.0 : BOOL;  (* Output Mapping *)
      RM53_STATE AT %ML1509 : ET_ROOM_STATE;
      RM53_BUZZER AT %MX81.0 : BOOL;  (* output mapping *)
      RM53_DIFF_PRESS AT %MD541 : REAL;  (* Input Mapping *)
      RM53_InAlarm AT %MX85.0 : BOOL;
      RM53_IsMute AT %MX85.1 : BOOL;
      RM53_GREEN_LED AT %MX84.0 : BOOL;  (* OUTPUT_MAPPING *)
      RM53_MODE_SWITCH AT %MX85.2 : BOOL;  (* Input Mapping *)
      RM53_STANDBY_LED AT %MX87.0 : BOOL;  (* Output Mapping *)
      RM53_RED_LED AT %MX86.0 : BOOL;  (* Output Mapping *)
      RM53_MUTE_BTN AT %MX85.3 : BOOL;  (* Input Mapping *)
      RM53_TRANSFER_DAMPER AT %MD543 : REAL;  (* OUTPUT MAPPING *)
      RM53_TRANSFER_DAMPER_ST AT %MD545 : REAL;  (* INPUT MAPPING *)
      RM59_DEPROX_SWITCH AT %MX92.3 : BOOL;  (* Input Mapping *)
      RM59_DEPROX_LED AT %MX92.0 : BOOL;  (* Output Mapping *)
      RM59_EXTRACT_DAMPER_ST AT %MX93.3 : BOOL;  (* Input Mapping *)
      RM59_EXTRACT_DAMPER AT %MX93.0 : BOOL;  (* Output Mapping *)
      RM59_SUPPLY_DAMPER_ST AT %MX98.3 : BOOL;  (* Input Mapping *)
      RM59_SUPPLY_DAMPER AT %MX98.0 : BOOL;  (* Output Mapping *)
      RM59_STATE AT %ML1510 : ET_ROOM_STATE;
      RM59_BUZZER AT %MX91.0 : BOOL;  (* output mapping *)
      RM59_DIFF_PRESS AT %MD546 : REAL;  (* Input Mapping *)
      RM59_InAlarm AT %MX95.0 : BOOL;
      RM59_IsMute AT %MX95.1 : BOOL;
      RM59_GREEN_LED AT %MX94.0 : BOOL;  (* OUTPUT_MAPPING *)
      RM59_MODE_SWITCH AT %MX95.2 : BOOL;  (* Input Mapping *)
      RM59_STANDBY_LED AT %MX97.0 : BOOL;  (* Output Mapping *)
      RM59_RED_LED AT %MX96.0 : BOOL;  (* Output Mapping *)
      RM59_MUTE_BTN AT %MX95.3 : BOOL;  (* Input Mapping *)
      RM59_TRANSFER_DAMPER AT %MD548 : REAL;  (* OUTPUT MAPPING *)
      RM59_TRANSFER_DAMPER_ST AT %MD550 : REAL;  (* INPUT MAPPING *)
      TOILET_EXTRACT_DAMPER_SS AT %MX100.0 : BOOL;  (* OUTPUT MAPPING *)
      TOILET_EXTRACT_DAMPER_ST AT %MX100.3 : BOOL;  (* Input Mapping *)
      FIRE_DAMPER AT %MX102.0 : BOOL;  (* Input Mapping *)
      DEPROX_SIGNAL1 AT %MX101.0 : BOOL;  (* 1 ROOM is in deprox mode *)
      DEPROX_SIGNAL2 AT %MX101.1 : BOOL;  (* 2 ROOM are in deprox mode *)
      DEPROX_SIGNAL3 AT %MX101.2 : BOOL;  (* 3 or more ROOM are in deprox mode *)
      RM44_SUPPLY_DAMPER_ST AT %MX103.0 : BOOL;  (* Input Mapping *)
      RM44_SUPPLY_DAMPER AT %MX103.1 : BOOL := TRUE;  (* Output Mapping *)
      RM6_DIFF_PRESS2 AT %MD551 : REAL;  (* Input Mapping *)
      RM6_DIFF_PRESS3 AT %MD553 : REAL;  (* Input Mapping *)
      RM71_ANTE_TO_RM_DIFF_PRESS AT %MD555 : REAL;  (* Input Mapping *)
      RM71_HALL_TO_ANTE_DIFF_PRESS AT %MD557 : REAL;  (* Input Mapping *)
      RM74_ANTEL_TO_RM_DIFF_PRESS AT %MD559 : REAL;  (* Input Mapping *)
      RM74_HALL_TO_ANTE_DIFF_PRESS AT %MD561 : REAL;  (* Input Mapping *)
      RM9_DIFF_PRESS2 AT %MD563 : REAL;  (* Input Mapping *)
      RM9_DIFF_PRESS3 AT %MD565 : REAL;  (* Input Mapping *)
      RM6_EXTRACT_DAMPER2 AT %MD581 : REAL;  (* Output Mapping *)
      RM6_EXTRACT_DAMPER2_ST AT %MD583 : REAL;  (* Input Mapping *)
      RM6_POSITIVE_MODE_SWITCH AT %MX19.4 : BOOL;  (* Input Mapping *)
      RM6_NEGATIVE_MODE_SWITCH AT %MX19.0 : BOOL;  (* Input Mapping *)
      RM6_POSITIVE_LED AT %MX19.1 : BOOL;  (* Output Mapping *)
      RM6_BOOSTER_FAN_SS AT %MX105.0 : BOOL;
      RM6_BOOSTER_FAN_SS_MD AT %MX105.1 : BOOL;
      RM6_BOOSTER_FAN_SS_OP AT %MX105.2 : BOOL;
      RM6_BOOSTER_FAN_SPD_MD AT %MX105.3 : BOOL;
      RM6_BOOSTER_FAN_SPD_OP AT %MD572 : REAL;
      RM6_BOOSTER_FAN_SPD AT %MD573 : REAL;
      RM6_BOOSTER_FAN_SPD_SP AT %MD576 : REAL;
      RM6_BOOSTER_FAN_STS AT %MX105.4 : BOOL;
      RM74_ADDITIONAL_TRANSFER_DAMPER AT %MD584 : REAL;  (* OUTPUT MAPPING *)
      RM74_ADDITIONAL_TRANSFER_DAMPER_ST AT %MD586 : REAL;  (* INPUT MAPPING *)
      RM119_ALARM_DELAY_SP AT %MW9001 : INT := 180;
      RM119_BUZZER_MANUAL AT %MX1.1 : BOOL := FALSE;
      RM119_BUZZER_MODE AT %MX1.2 : BOOL := TRUE;  (* 1 = AUTO 0 = MANUAL *)
      RM119_DIFF_PRESS_SP AT %MD502 : REAL := 8;
      RM119_STANDBY_LED_MANUAL AT %MX7.1 : BOOL := FALSE;
      RM119_STANDBY_LED_MODE AT %MX7.2 : BOOL := TRUE;  (* 1 = AUTO 0 = MANUAL *)
      RM119_GREEN_LED_MANUAL AT %MX4.1 : BOOL := FALSE;
      RM119_GREEN_LED_MODE AT %MX4.2 : BOOL := TRUE;  (* 1 = AUTO 0 = MANUAL *)
      RM119_RED_LED_MANUAL AT %MX6.1 : BOOL := FALSE;
      RM119_RED_LED_MODE AT %MX6.2 : BOOL := TRUE;  (* 1 = AUTO 0 = MANUAL *)
      RM119_DEPROX_LED_MANUAL AT %MX2.1 : BOOL;
      RM119_DEPROX_LED_MODE AT %MX2.2 : BOOL := TRUE;  (* 1 = AUTO 0 = MANUAL *)
      RM119_EXTRACT_DAMPER_MANUAL AT %MX3.1 : BOOL := FALSE;
      RM119_EXTRACT_DAMPER_MODE AT %MX3.2 : BOOL := TRUE;  (* 1 = AUTO 0 = MANUAL *)
      RM119_SUPPLY_DAMPER_MANUAL AT %MX8.1 : BOOL := FALSE;
      RM119_SUPPLY_DAMPER_MODE AT %MX8.2 : BOOL := TRUE;  (* 1 = AUTO 0 = MANUAL *)
      RM119_TRANSFER_DAMPER_SP AT %MD504 : REAL := 75;
      RM6_ALARM_DELAY_SP AT %MW9002 : INT := 180;
      RM6_BUZZER_MANUAL AT %MX11.1 : BOOL := FALSE;
      RM6_BUZZER_MODE AT %MX11.2 : BOOL := TRUE;  (* 1 = AUTO 0 = MANUAL *)
      RM6_DIFF_PRESS_SP1 AT %MD507 : REAL := 8;
      RM6_STANDBY_LED_MANUAL AT %MX17.1 : BOOL := FALSE;
      RM6_STANDBY_LED_MODE AT %MX17.2 : BOOL := TRUE;  (* 1 = AUTO 0 = MANUAL *)
      RM6_GREEN_LED_MANUAL AT %MX14.1 : BOOL := FALSE;
      RM6_GREEN_LED_MODE AT %MX14.2 : BOOL := TRUE;  (* 1 = AUTO 0 = MANUAL *)
      RM6_RED_LED_MANUAL AT %MX16.1 : BOOL := FALSE;
      RM6_RED_LED_MODE AT %MX16.2 : BOOL := TRUE;  (* 1 = AUTO 0 = MANUAL *)
      RM6_DEPROX_LED_MANUAL AT %MX12.1 : BOOL;
      RM6_DEPROX_LED_MODE AT %MX12.2 : BOOL := TRUE;  (* 1 = AUTO 0 = MANUAL *)
      RM6_EXTRACT_DAMPER1_MANUAL AT %MD579 : REAL := 100;
      RM6_EXTRACT_DAMPER1_MODE AT %MX13.2 : BOOL := TRUE;  (* 1 = AUTO 0 = MANUAL *)
      RM6_SUPPLY_DAMPER_MANUAL AT %MD570 : REAL;
      RM6_SUPPLY_DAMPER_MODE AT %MX18.2 : BOOL := TRUE;  (* 1 = AUTO 0 = MANUAL *)
      RM6_TRANSFER_DAMPER_SP AT %MD509 : REAL := 75;
      RM71_ALARM_DELAY_SP AT %MW9003 : INT := 180;
      RM71_BUZZER_MANUAL AT %MX21.1 : BOOL := FALSE;
      RM71_BUZZER_MODE AT %MX21.2 : BOOL := TRUE;  (* 1 = AUTO 0 = MANUAL *)
      RM71_HALL_TO_RM_DIFF_PRESS_SP AT %MD512 : REAL := 8;
      RM71_STANDBY_LED_MANUAL AT %MX27.1 : BOOL := FALSE;
      RM71_STANDBY_LED_MODE AT %MX27.2 : BOOL := TRUE;  (* 1 = AUTO 0 = MANUAL *)
      RM71_GREEN_LED_MANUAL AT %MX24.1 : BOOL := FALSE;
      RM71_GREEN_LED_MODE AT %MX24.2 : BOOL := TRUE;  (* 1 = AUTO 0 = MANUAL *)
      RM71_RED_LED_MANUAL AT %MX26.1 : BOOL := FALSE;
      RM71_RED_LED_MODE AT %MX26.2 : BOOL := TRUE;  (* 1 = AUTO 0 = MANUAL *)
      RM71_DEPROX_LED_MANUAL AT %MX22.1 : BOOL;
      RM71_DEPROX_LED_MODE AT %MX22.2 : BOOL := TRUE;  (* 1 = AUTO 0 = MANUAL *)
      RM71_EXTRACT_DAMPER_MANUAL AT %MX23.1 : BOOL := FALSE;
      RM71_EXTRACT_DAMPER_MODE AT %MX23.2 : BOOL := TRUE;  (* 1 = AUTO 0 = MANUAL *)
      RM71_SUPPLY_DAMPER_MANUAL AT %MX28.1 : BOOL := FALSE;
      RM71_SUPPLY_DAMPER_MODE AT %MX28.2 : BOOL := TRUE;  (* 1 = AUTO 0 = MANUAL *)
      RM71_TRANSFER_DAMPER_SP AT %MD514 : REAL := 75;  (* OUTPUT MAPPING *)
      RM74_ALARM_DELAY_SP AT %MW9004 : INT := 180;
      RM74_BUZZER_MANUAL AT %MX31.1 : BOOL := FALSE;
      RM74_BUZZER_MODE AT %MX31.2 : BOOL := TRUE;  (* 1 = AUTO 0 = MANUAL *)
      RM74_HALL_TO_RM_DIFF_PRESS_SP AT %MD517 : REAL := 8;
      RM74_STANDBY_LED_MANUAL AT %MX37.1 : BOOL := FALSE;
      RM74_STANDBY_LED_MODE AT %MX37.2 : BOOL := TRUE;  (* 1 = AUTO 0 = MANUAL *)
      RM74_GREEN_LED_MANUAL AT %MX34.1 : BOOL := FALSE;
      RM74_GREEN_LED_MODE AT %MX34.2 : BOOL := TRUE;  (* 1 = AUTO 0 = MANUAL *)
      RM74_RED_LED_MANUAL AT %MX36.1 : BOOL := FALSE;
      RM74_RED_LED_MODE AT %MX36.2 : BOOL := TRUE;  (* 1 = AUTO 0 = MANUAL *)
      RM74_DEPROX_LED_MANUAL AT %MX32.1 : BOOL;
      RM74_DEPROX_LED_MODE AT %MX32.2 : BOOL := TRUE;  (* 1 = AUTO 0 = MANUAL *)
      RM74_EXTRACT_DAMPER_MANUAL AT %MX33.1 : BOOL := FALSE;
      RM74_EXTRACT_DAMPER_MODE AT %MX33.2 : BOOL := TRUE;  (* 1 = AUTO 0 = MANUAL *)
      RM74_SUPPLY_DAMPER_MANUAL AT %MX38.1 : BOOL := FALSE;
      RM74_SUPPLY_DAMPER_MODE AT %MX38.2 : BOOL := TRUE;  (* 1 = AUTO 0 = MANUAL *)
      RM74_TRANSFER_DAMPER_SP AT %MD519 : REAL := 75;
      RM9_ALARM_DELAY_SP AT %MW9005 : INT := 180;
      RM9_BUZZER_MANUAL AT %MX41.1 : BOOL := FALSE;
      RM9_BUZZER_MODE AT %MX41.2 : BOOL := TRUE;  (* 1 = AUTO 0 = MANUAL *)
      RM9_DIFF_PRESS_SP1 AT %MD522 : REAL := 8;
      RM9_STANDBY_LED_MANUAL AT %MX47.1 : BOOL := FALSE;
      RM9_STANDBY_LED_MODE AT %MX47.2 : BOOL := TRUE;  (* 1 = AUTO 0 = MANUAL *)
      RM9_GREEN_LED_MANUAL AT %MX44.1 : BOOL := FALSE;
      RM9_GREEN_LED_MODE AT %MX44.2 : BOOL := TRUE;  (* 1 = AUTO 0 = MANUAL *)
      RM9_RED_LED_MANUAL AT %MX46.1 : BOOL := FALSE;
      RM9_RED_LED_MODE AT %MX46.2 : BOOL := TRUE;  (* 1 = AUTO 0 = MANUAL *)
      RM9_DEPROX_LED_MANUAL AT %MX42.1 : BOOL;
      RM9_DEPROX_LED_MODE AT %MX42.2 : BOOL := TRUE;  (* 1 = AUTO 0 = MANUAL *)
      RM9_EXTRACT_DAMPER_MANUAL AT %MX43.1 : BOOL := FALSE;
      RM9_EXTRACT_DAMPER_MODE AT %MX43.2 : BOOL := TRUE;  (* 1 = AUTO 0 = MANUAL *)
      RM9_SUPPLY_DAMPER_MANUAL AT %MX48.1 : BOOL := FALSE;
      RM9_SUPPLY_DAMPER_MODE AT %MX48.2 : BOOL := TRUE;  (* 1 = AUTO 0 = MANUAL *)
      RM9_TRANSFER_DAMPER_SP AT %MD524 : REAL := 75;
      RM44_3_ALARM_DELAY_SP AT %MW9006 : INT := 180;
      RM44_3_BUZZER_MANUAL AT %MX51.1 : BOOL := FALSE;
      RM44_3_BUZZER_MODE AT %MX51.2 : BOOL := TRUE;  (* 1 = AUTO 0 = MANUAL *)
      RM44_3_DIFF_PRESS_SP AT %MD527 : REAL := 8;
      RM44_3_STANDBY_LED_MANUAL AT %MX57.1 : BOOL := FALSE;
      RM44_3_STANDBY_LED_MODE AT %MX57.2 : BOOL := TRUE;  (* 1 = AUTO 0 = MANUAL *)
      RM44_3_GREEN_LED_MANUAL AT %MX54.1 : BOOL := FALSE;
      RM44_3_GREEN_LED_MODE AT %MX54.2 : BOOL := TRUE;  (* 1 = AUTO 0 = MANUAL *)
      RM44_3_RED_LED_MANUAL AT %MX56.1 : BOOL := FALSE;
      RM44_3_RED_LED_MODE AT %MX56.2 : BOOL := TRUE;  (* 1 = AUTO 0 = MANUAL *)
      RM44_3_DEPROX_LED_MANUAL AT %MX52.1 : BOOL;
      RM44_3_DEPROX_LED_MODE AT %MX52.2 : BOOL := TRUE;  (* 1 = AUTO 0 = MANUAL *)
      RM44_3_EXTRACT_DAMPER_MANUAL AT %MX53.1 : BOOL := FALSE;
      RM44_3_EXTRACT_DAMPER_MODE AT %MX53.2 : BOOL := TRUE;  (* 1 = AUTO 0 = MANUAL *)
      RM44_3_SUPPLY_DAMPER_MANUAL AT %MX58.1 : BOOL := FALSE;
      RM44_3_SUPPLY_DAMPER_MODE AT %MX58.2 : BOOL := TRUE;  (* 1 = AUTO 0 = MANUAL *)
      RM44_3_TRANSFER_DAMPER_SP AT %MD529 : REAL := 75;
      RM51_ALARM_DELAY_SP AT %MW9007 : INT := 180;
      RM51_BUZZER_MANUAL AT %MX61.1 : BOOL := FALSE;
      RM51_BUZZER_MODE AT %MX61.2 : BOOL := TRUE;  (* 1 = AUTO 0 = MANUAL *)
      RM51_DIFF_PRESS_SP AT %MD532 : REAL := 8;
      RM51_STANDBY_LED_MANUAL AT %MX67.1 : BOOL := FALSE;
      RM51_STANDBY_LED_MODE AT %MX67.2 : BOOL := TRUE;  (* 1 = AUTO 0 = MANUAL *)
      RM51_GREEN_LED_MANUAL AT %MX64.1 : BOOL := FALSE;
      RM51_GREEN_LED_MODE AT %MX64.2 : BOOL := TRUE;  (* 1 = AUTO 0 = MANUAL *)
      RM51_RED_LED_MANUAL AT %MX66.1 : BOOL := FALSE;
      RM51_RED_LED_MODE AT %MX66.2 : BOOL := TRUE;  (* 1 = AUTO 0 = MANUAL *)
      RM51_DEPROX_LED_MANUAL AT %MX62.1 : BOOL;
      RM51_DEPROX_LED_MODE AT %MX62.2 : BOOL := TRUE;  (* 1 = AUTO 0 = MANUAL *)
      RM51_EXTRACT_DAMPER_MANUAL AT %MX63.1 : BOOL := FALSE;
      RM51_EXTRACT_DAMPER_MODE AT %MX63.2 : BOOL := TRUE;  (* 1 = AUTO 0 = MANUAL *)
      RM51_SUPPLY_DAMPER_MANUAL AT %MX68.1 : BOOL := FALSE;
      RM51_SUPPLY_DAMPER_MODE AT %MX68.2 : BOOL := TRUE;  (* 1 = AUTO 0 = MANUAL *)
      RM51_TRANSFER_DAMPER_SP AT %MD534 : REAL := 75;
      RM52_ALARM_DELAY_SP AT %MW9008 : INT := 180;
      RM52_BUZZER_MANUAL AT %MX71.1 : BOOL := FALSE;
      RM52_BUZZER_MODE AT %MX71.2 : BOOL := TRUE;  (* 1 = AUTO 0 = MANUAL *)
      RM52_DIFF_PRESS_SP AT %MD537 : REAL := 8;
      RM52_STANDBY_LED_MANUAL AT %MX77.1 : BOOL := FALSE;
      RM52_STANDBY_LED_MODE AT %MX77.2 : BOOL := TRUE;  (* 1 = AUTO 0 = MANUAL *)
      RM52_GREEN_LED_MANUAL AT %MX74.1 : BOOL := FALSE;
      RM52_GREEN_LED_MODE AT %MX74.2 : BOOL := TRUE;  (* 1 = AUTO 0 = MANUAL *)
      RM52_RED_LED_MANUAL AT %MX76.1 : BOOL := FALSE;
      RM52_RED_LED_MODE AT %MX76.2 : BOOL := TRUE;  (* 1 = AUTO 0 = MANUAL *)
      RM52_DEPROX_LED_MANUAL AT %MX72.1 : BOOL;
      RM52_DEPROX_LED_MODE AT %MX72.2 : BOOL := TRUE;  (* 1 = AUTO 0 = MANUAL *)
      RM52_EXTRACT_DAMPER_MANUAL AT %MX73.1 : BOOL := FALSE;
      RM52_EXTRACT_DAMPER_MODE AT %MX73.2 : BOOL := TRUE;  (* 1 = AUTO 0 = MANUAL *)
      RM52_SUPPLY_DAMPER_MANUAL AT %MX78.1 : BOOL := FALSE;
      RM52_SUPPLY_DAMPER_MODE AT %MX78.2 : BOOL := TRUE;  (* 1 = AUTO 0 = MANUAL *)
      RM52_TRANSFER_DAMPER_SP AT %MD539 : REAL := 75;
      RM53_ALARM_DELAY_SP AT %MW9009 : INT := 180;
      RM53_BUZZER_MANUAL AT %MX81.1 : BOOL := FALSE;
      RM53_BUZZER_MODE AT %MX81.2 : BOOL := TRUE;  (* 1 = AUTO 0 = MANUAL *)
      RM53_DIFF_PRESS_SP AT %MD542 : REAL := 8;
      RM53_STANDBY_LED_MANUAL AT %MX87.1 : BOOL := FALSE;
      RM53_STANDBY_LED_MODE AT %MX87.2 : BOOL := TRUE;  (* 1 = AUTO 0 = MANUAL *)
      RM53_GREEN_LED_MANUAL AT %MX84.1 : BOOL := FALSE;
      RM53_GREEN_LED_MODE AT %MX84.2 : BOOL := TRUE;  (* 1 = AUTO 0 = MANUAL *)
      RM53_RED_LED_MANUAL AT %MX86.1 : BOOL := FALSE;
      RM53_RED_LED_MODE AT %MX86.2 : BOOL := TRUE;  (* 1 = AUTO 0 = MANUAL *)
      RM53_DEPROX_LED_MANUAL AT %MX82.1 : BOOL;
      RM53_DEPROX_LED_MODE AT %MX82.2 : BOOL := TRUE;  (* 1 = AUTO 0 = MANUAL *)
      RM53_EXTRACT_DAMPER_MANUAL AT %MX83.1 : BOOL := FALSE;
      RM53_EXTRACT_DAMPER_MODE AT %MX83.2 : BOOL := TRUE;  (* 1 = AUTO 0 = MANUAL *)
      RM53_SUPPLY_DAMPER_MANUAL AT %MX88.1 : BOOL := FALSE;
      RM53_SUPPLY_DAMPER_MODE AT %MX88.2 : BOOL := TRUE;  (* 1 = AUTO 0 = MANUAL *)
      RM53_TRANSFER_DAMPER_SP AT %MD544 : REAL := 75;
      RM59_ALARM_DELAY_SP AT %MW9010 : INT := 180;
      RM59_BUZZER_MANUAL AT %MX91.1 : BOOL := FALSE;
      RM59_BUZZER_MODE AT %MX91.2 : BOOL := TRUE;  (* 1 = AUTO 0 = MANUAL *)
      RM59_DIFF_PRESS_SP AT %MD547 : REAL := 8;
      RM59_STANDBY_LED_MANUAL AT %MX97.1 : BOOL := FALSE;
      RM59_STANDBY_LED_MODE AT %MX97.2 : BOOL := TRUE;  (* 1 = AUTO 0 = MANUAL *)
      RM59_GREEN_LED_MANUAL AT %MX94.1 : BOOL := FALSE;
      RM59_GREEN_LED_MODE AT %MX94.2 : BOOL := TRUE;  (* 1 = AUTO 0 = MANUAL *)
      RM59_RED_LED_MANUAL AT %MX96.1 : BOOL := FALSE;
      RM59_RED_LED_MODE AT %MX96.2 : BOOL := TRUE;  (* 1 = AUTO 0 = MANUAL *)
      RM59_DEPROX_LED_MANUAL AT %MX92.1 : BOOL;
      RM59_DEPROX_LED_MODE AT %MX92.2 : BOOL := TRUE;  (* 1 = AUTO 0 = MANUAL *)
      RM59_EXTRACT_DAMPER_MANUAL AT %MX93.1 : BOOL := FALSE;
      RM59_EXTRACT_DAMPER_MODE AT %MX93.2 : BOOL := TRUE;  (* 1 = AUTO 0 = MANUAL *)
      RM59_SUPPLY_DAMPER_MANUAL AT %MX98.1 : BOOL := FALSE;
      RM59_SUPPLY_DAMPER_MODE AT %MX98.2 : BOOL := TRUE;  (* 1 = AUTO 0 = MANUAL *)
      RM59_TRANSFER_DAMPER_SP AT %MD549 : REAL := 75;
      TOILET_EXTRACT_DAMPER_SS_MANUAL AT %MX100.1 : BOOL := FALSE;
      TOILET_EXTRACT_DAMPER_SS_MODE AT %MX100.2 : BOOL := TRUE;  (* 1 = AUTO 0 = MANUAL *)
      RM6_DIFF_PRESS_SP2 AT %MD552 : REAL := 8;
      RM6_DIFF_PRESS_SP3 AT %MD554 : REAL := 8;
      RM71_ANTE_TO_RM_DIFF_PRESS_SP AT %MD556 : REAL := 8;
      RM71_HALL_TO_ANTE_DIFF_PRESS_SP AT %MD558 : REAL := 8;
      RM74_ANTEL_TO_RM_DIFF_PRESS_SP AT %MD560 : REAL := 8;
      RM74_HALL_TO_ANTE_DIFF_PRESS_SP AT %MD562 : REAL := 8;
      RM9_DIFF_PRESS_SP2 AT %MD564 : REAL := 8;
      RM9_DIFF_PRESS_SP3 AT %MD566 : REAL := 8;
      RM6_EXTRACT_DAMPER2_MANUAL AT %MD582 : REAL := 100;
      RM6_EXTRACT_DAMPER2_MODE AT %MX13.6 : BOOL := TRUE;  (* 1 = AUTO 0 = MANUAL *)
      RM6_POSITIVE_LED_MANUAL AT %MX19.2 : BOOL := FALSE;
      RM6_POSITIVE_LED_MODE AT %MX19.3 : BOOL := TRUE;  (* 1 = AUTO 0 = MANUAL *)
      RM74_ADDITIONAL_TRANSFER_DAMPER_SP AT %MD585 : REAL := 75;
    END_VAR
    TASK MAST(INTERVAL := T#20ms, PRIORITY := 15);
    PROGRAM INPUT_MAPPING WITH MAST : INPUT_MAPPING;
    PROGRAM RM71_DEPROX WITH MAST : RM71_DEPROX;
    PROGRAM RM71_STATUS WITH MAST : RM71_STATUS;
    PROGRAM RM74_DEPROX WITH MAST : RM74_DEPROX;
    PROGRAM RM74_STATUS WITH MAST : RM74_STATUS;
    PROGRAM DEPROX_SIGNAL WITH MAST : DEPROX_SIGNAL;
    PROGRAM OUTPUT_MAPPING WITH MAST : OUTPUT_MAPPING;
  END_RESOURCE
END_CONFIGURATION

CONFIGURATION IO_Bus
END_CONFIGURATION

CONFIGURATION Module_1
END_CONFIGURATION

CONFIGURATION Module_3
END_CONFIGURATION

CONFIGURATION Module_4
END_CONFIGURATION

CONFIGURATION COM_Bus
END_CONFIGURATION

CONFIGURATION Ethernet_1
END_CONFIGURATION

CONFIGURATION Serial_Line_1
END_CONFIGURATION

CONFIGURATION Machine_Expert_Network_Manager
END_CONFIGURATION

CONFIGURATION CAN_1
END_CONFIGURATION
